LIN {X 0,Y 354.586,Z 442.804,A -85,B 0,C 180,E1 -14686.804,E2 -14686.804} C_VEL
LIN {X 0,Y 350.796,Z 438.924,A -85,B 0,C 180,E1 -14687.678,E2 -14687.678} C_VEL
LIN {X 0,Y 348.706,Z 436.523,A -85,B 0,C 180,E1 -14688.15,E2 -14688.15} C_VEL
LIN {X 0,Y 345.386,Z 432.719,A -85,B 0,C 180,E1 -14688.87,E2 -14688.87} C_VEL
LIN {X 0,Y 343.539,Z 430.553,A -85,B 0,C 180,E1 -14689.252,E2 -14689.252} C_VEL
LIN {X 0,Y 340.657,Z 426.868,A -85,B 0,C 180,E1 -14689.842,E2 -14689.842} C_VEL
LIN {X 0,Y 337.415,Z 422.834,A -85,B 0,C 180,E1 -14690.475,E2 -14690.475} C_VEL
LIN {X 0,Y 336.252,Z 421.04,A -85,B 0,C 180,E1 -14690.703,E2 -14690.703} C_VEL
LIN {X 0,Y 334.391,Z 418.724,A -85,B 0,C 180,E1 -14691.054,E2 -14691.054} C_VEL
LIN {X 0,Y 333.681,Z 416.421,A -85,B 0,C 180,E1 -14691.256,E2 -14691.256} C_VEL
LIN {X 0,Y 333.714,Z 416.415,A -85,B 0,C 180,E1 -14695.101,E2 -14695.101} C_VEL
LIN {X 0,Y 333.711,Z 416.417,A -85,B 0,C 180,E1 -14697.809,E2 -14697.809} C_VEL
LIN {X 0,Y 333.685,Z 416.417,A -85,B 0,C 180,E1 -14700.363,E2 -14700.363} C_VEL
LIN {X 0,Y 333.668,Z 416.419,A -85,B 0,C 180,E1 -14704.658,E2 -14704.658} C_VEL
LIN {X 0,Y 333.648,Z 416.425,A -85,B 0,C 180,E1 -14707.651,E2 -14707.651} C_VEL
LIN {X 0,Y 333.64,Z 416.423,A -85,B 0,C 180,E1 -14710.767,E2 -14710.767} C_VEL
LIN {X 0,Y 333.619,Z 416.425,A -85,B 0,C 180,E1 -14714.256,E2 -14714.256} C_VEL
LIN {X 0,Y 333.635,Z 416.425,A -85,B 0,C 180,E1 -14717.618,E2 -14717.618} C_VEL
LIN {X 0,Y 333.645,Z 416.427,A -85,B 0,C 180,E1 -14721.202,E2 -14721.202} C_VEL
LIN {X 0,Y 333.669,Z 416.419,A -85,B 0,C 180,E1 -14723.861,E2 -14723.861} C_VEL
LIN {X 0,Y 333.636,Z 416.425,A -85,B 0,C 180,E1 -14727.413,E2 -14727.413} C_VEL
LIN {X 0,Y 333.704,Z 416.42,A -85,B 0,C 180,E1 -14731.028,E2 -14731.028} C_VEL
LIN {X 0,Y 333.705,Z 416.417,A -85,B 0,C 180,E1 -14734.698,E2 -14734.698} C_VEL
LIN {X 0,Y 333.712,Z 416.413,A -85,B 0,C 180,E1 -14737.914,E2 -14737.914} C_VEL
LIN {X 0,Y 333.697,Z 416.414,A -85,B 0,C 180,E1 -14739.932,E2 -14739.932} C_VEL
LIN {X 0,Y 333.086,Z 416.496,A -85,B 0,C 180,E1 -14740.94,E2 -14740.94} C_VEL
LIN {X 0,Y 330.26,Z 416.849,A -85,B 0,C 180,E1 -14742.579,E2 -14742.579} C_VEL
LIN {X 0,Y 327.845,Z 417.15,A -85,B 0,C 180,E1 -14743.907,E2 -14743.907} C_VEL
LIN {X 0,Y 326.824,Z 417.275,A -85,B 0,C 180,E1 -14744.934,E2 -14744.934} C_VEL
LIN {X 0,Y 326.75,Z 417.281,A -85,B 0,C 180,E1 -14745.283,E2 -14745.283} C_VEL
LIN {X 0,Y 326.762,Z 417.283,A -85,B 0,C 180,E1 -14748.839,E2 -14748.839} C_VEL
LIN {X 0,Y 326.951,Z 417.26,A -85,B 0,C 180,E1 -14752.59,E2 -14752.59} C_VEL
LIN {X 0,Y 326.771,Z 417.278,A -85,B 0,C 180,E1 -14755.065,E2 -14755.065} C_VEL
LIN {X 0,Y 327.041,Z 417.239,A -85,B 0,C 180,E1 -14757.537,E2 -14757.537} C_VEL
LIN {X 0,Y 327.191,Z 417.223,A -85,B 0,C 180,E1 -14760.001,E2 -14760.001} C_VEL
LIN {X 0,Y 327.041,Z 417.249,A -85,B 0,C 180,E1 -14762.464,E2 -14762.464} C_VEL
LIN {X 0,Y 326.983,Z 417.255,A -85,B 0,C 180,E1 -14766.17,E2 -14766.17} C_VEL
LIN {X 0,Y 326.799,Z 417.276,A -85,B 0,C 180,E1 -14769.907,E2 -14769.907} C_VEL
LIN {X 0,Y 326.753,Z 417.281,A -85,B 0,C 180,E1 -14773.686,E2 -14773.686} C_VEL
LIN {X 0,Y 326.694,Z 417.288,A -85,B 0,C 180,E1 -14777.529,E2 -14777.529} C_VEL
LIN {X 0,Y 326.653,Z 417.298,A -85,B 0,C 180,E1 -14780.136,E2 -14780.136} C_VEL
LIN {X 0,Y 326.644,Z 417.3,A -85,B 0,C 180,E1 -14784.13,E2 -14784.13} C_VEL
LIN {X 0,Y 326.681,Z 417.29,A -85,B 0,C 180,E1 -14786.859,E2 -14786.859} C_VEL
LIN {X 0,Y 326.638,Z 417.298,A -85,B 0,C 180,E1 -14790.613,E2 -14790.613} C_VEL
LIN {X 0,Y 326.606,Z 417.305,A -85,B 0,C 180,E1 -14794.02,E2 -14794.02} C_VEL
LIN {X 0,Y 326.683,Z 417.655,A -85,B 0,C 180,E1 -14795.511,E2 -14795.511} C_VEL
LIN {X 0,Y 327.038,Z 420.312,A -85,B 0,C 180,E1 -14799.32,E2 -14799.32} C_VEL
LIN {X 0,Y 327.48,Z 423.224,A -85,B 0,C 180,E1 -14803.143,E2 -14803.143} C_VEL
LIN {X 0,Y 327.639,Z 424.827,A -85,B 0,C 180,E1 -14805.062,E2 -14805.062} C_VEL
LIN {X 0,Y 327.663,Z 427.715,A -85,B 0,C 180,E1 -14808.325,E2 -14808.325} C_VEL
LIN {X 0,Y 327.32,Z 430.741,A -85,B 0,C 180,E1 -14811.49,E2 -14811.49} C_VEL
LIN {X 0,Y 326.883,Z 434.094,A -85,B 0,C 180,E1 -14814.787,E2 -14814.787} C_VEL
LIN {X 0,Y 326.537,Z 436.909,A -85,B 0,C 180,E1 -14817.448,E2 -14817.448} C_VEL
LIN {X 0,Y 326.123,Z 440.042,A -85,B 0,C 180,E1 -14820.288,E2 -14820.288} C_VEL
LIN {X 0,Y 325.778,Z 443.169,A -85,B 0,C 180,E1 -14823.062,E2 -14823.062} C_VEL
LIN {X 0,Y 325.536,Z 446.331,A -85,B 0,C 180,E1 -14825.784,E2 -14825.784} C_VEL
LIN {X 0,Y 325.333,Z 448.523,A -85,B 0,C 180,E1 -14827.658,E2 -14827.658} C_VEL
LIN {X 0,Y 328.277,Z 460.951,A -85,B 0,C 180,E1 -14828.388,E2 -14828.388} C_VEL
LIN {X 0,Y 330.744,Z 474.544,A -85,B 0,C 180,E1 -14829.4,E2 -14829.4} C_VEL
LIN {X 0,Y 331.996,Z 485.066,A -85,B 0,C 180,E1 -14830.364,E2 -14830.364} C_VEL
LIN {X 0,Y 332.325,Z 489.987,A -85,B 0,C 180,E1 -14830.866,E2 -14830.866} C_VEL
LIN {X 0,Y 330.84,Z 502.177,A -85,B 0,C 180,E1 -14832.22,E2 -14832.22} C_VEL
LIN {X 0,Y 329.853,Z 509.927,A -85,B 0,C 180,E1 -14833.284,E2 -14833.284} C_VEL
LIN {X 0,Y 328.869,Z 517.509,A -85,B 0,C 180,E1 -14834.521,E2 -14834.521} C_VEL
LIN {X 0,Y 327.798,Z 525.266,A -85,B 0,C 180,E1 -14836.043,E2 -14836.043} C_VEL
LIN {X 0,Y 326.796,Z 531.801,A -85,B 0,C 180,E1 -14837.581,E2 -14837.581} C_VEL
LIN {X 0,Y 326.23,Z 536.304,A -85,B 0,C 180,E1 -14838.82,E2 -14838.82} C_VEL
LIN {X 0,Y 325.601,Z 541.798,A -85,B 0,C 180,E1 -14840.684,E2 -14840.684} C_VEL
LIN {X 0,Y 325.159,Z 546.124,A -85,B 0,C 180,E1 -14842.549,E2 -14842.549} C_VEL
LIN {X 0,Y 324.906,Z 549.205,A -85,B 0,C 180,E1 -14844.285,E2 -14844.285} C_VEL
LIN {X 0,Y 324.902,Z 551.682,A -85,B 0,C 180,E1 -14846.279,E2 -14846.279} C_VEL
LIN {X 0,Y 324.838,Z 552.74,A -85,B 0,C 180,E1 -14847.52,E2 -14847.52} C_VEL
LIN {X 0,Y 324.823,Z 553.329,A -85,B 0,C 180,E1 -14848.76,E2 -14848.76} C_VEL
LIN {X 0,Y 324.873,Z 553.485,A -85,B 0,C 180,E1 -14850,E2 -14850} C_VEL
LIN {X 0,Y 324.823,Z 553.329,A -85,B 0,C 180,E1 -14851.24,E2 -14851.24} C_VEL
LIN {X 0,Y 324.838,Z 552.74,A -85,B 0,C 180,E1 -14852.48,E2 -14852.48} C_VEL
LIN {X 0,Y 324.892,Z 550.292,A -85,B 0,C 180,E1 -14854.964,E2 -14854.964} C_VEL
LIN {X 0,Y 325.047,Z 547.341,A -85,B 0,C 180,E1 -14856.83,E2 -14856.83} C_VEL
LIN {X 0,Y 325.423,Z 543.352,A -85,B 0,C 180,E1 -14858.695,E2 -14858.695} C_VEL
LIN {X 0,Y 325.993,Z 538.221,A -85,B 0,C 180,E1 -14860.559,E2 -14860.559} C_VEL
LIN {X 0,Y 326.648,Z 532.957,A -85,B 0,C 180,E1 -14862.109,E2 -14862.109} C_VEL
LIN {X 0,Y 327.582,Z 526.642,A -85,B 0,C 180,E1 -14863.65,E2 -14863.65} C_VEL
LIN {X 0,Y 328.363,Z 520.689,A -85,B 0,C 180,E1 -14864.882,E2 -14864.882} C_VEL
LIN {X 0,Y 329.338,Z 513.197,A -85,B 0,C 180,E1 -14866.199,E2 -14866.199} C_VEL
LIN {X 0,Y 330.33,Z 505.58,A -85,B 0,C 180,E1 -14867.329,E2 -14867.329} C_VEL
LIN {X 0,Y 331.467,Z 497.071,A -85,B 0,C 180,E1 -14868.384,E2 -14868.384} C_VEL
LIN {X 0,Y 332.302,Z 489.987,A -85,B 0,C 180,E1 -14869.136,E2 -14869.136} C_VEL
LIN {X 0,Y 331.418,Z 479.637,A -85,B 0,C 180,E1 -14870.149,E2 -14870.149} C_VEL
LIN {X 0,Y 329.995,Z 469.715,A -85,B 0,C 180,E1 -14870.978,E2 -14870.978} C_VEL
LIN {X 0,Y 327.939,Z 459.393,A -85,B 0,C 180,E1 -14871.708,E2 -14871.708} C_VEL
LIN {X 0,Y 325.333,Z 448.523,A -85,B 0,C 180,E1 -14872.342,E2 -14872.342} C_VEL
LIN {X 0,Y 325.64,Z 444.744,A -85,B 0,C 180,E1 -14875.571,E2 -14875.571} C_VEL
LIN {X 0,Y 325.925,Z 441.591,A -85,B 0,C 180,E1 -14878.319,E2 -14878.319} C_VEL
LIN {X 0,Y 326.33,Z 438.464,A -85,B 0,C 180,E1 -14881.122,E2 -14881.122} C_VEL
LIN {X 0,Y 326.71,Z 435.355,A -85,B 0,C 180,E1 -14884.006,E2 -14884.006} C_VEL
LIN {X 0,Y 327.172,Z 431.885,A -85,B 0,C 180,E1 -14887.363,E2 -14887.363} C_VEL
LIN {X 0,Y 327.499,Z 429.209,A -85,B 0,C 180,E1 -14890.074,E2 -14890.074} C_VEL
LIN {X 0,Y 327.671,Z 426.322,A -85,B 0,C 180,E1 -14893.176,E2 -14893.176} C_VEL
LIN {X 0,Y 327.613,Z 424.686,A -85,B 0,C 180,E1 -14895.065,E2 -14895.065} C_VEL
LIN {X 0,Y 327.24,Z 421.707,A -85,B 0,C 180,E1 -14898.735,E2 -14898.735} C_VEL
LIN {X 0,Y 326.823,Z 418.85,A -85,B 0,C 180,E1 -14902.715,E2 -14902.715} C_VEL
LIN {X 0,Y 326.637,Z 417.429,A -85,B 0,C 180,E1 -14904.845,E2 -14904.845} C_VEL
LIN {X 0,Y 326.612,Z 417.303,A -85,B 0,C 180,E1 -14907.455,E2 -14907.455} C_VEL
LIN {X 0,Y 326.658,Z 417.295,A -85,B 0,C 180,E1 -14910.34,E2 -14910.34} C_VEL
LIN {X 0,Y 326.686,Z 417.29,A -85,B 0,C 180,E1 -14914.515,E2 -14914.515} C_VEL
LIN {X 0,Y 326.614,Z 417.299,A -85,B 0,C 180,E1 -14918.542,E2 -14918.542} C_VEL
LIN {X 0,Y 326.74,Z 417.283,A -85,B 0,C 180,E1 -14921.177,E2 -14921.177} C_VEL
LIN {X 0,Y 326.758,Z 417.283,A -85,B 0,C 180,E1 -14925.432,E2 -14925.432} C_VEL
LIN {X 0,Y 326.763,Z 417.279,A -85,B 0,C 180,E1 -14928.838,E2 -14928.838} C_VEL
LIN {X 0,Y 326.952,Z 417.255,A -85,B 0,C 180,E1 -14932.589,E2 -14932.589} C_VEL
LIN {X 0,Y 326.771,Z 417.28,A -85,B 0,C 180,E1 -14935.064,E2 -14935.064} C_VEL
LIN {X 0,Y 327.041,Z 417.249,A -85,B 0,C 180,E1 -14937.536,E2 -14937.536} C_VEL
LIN {X 0,Y 327.191,Z 417.223,A -85,B 0,C 180,E1 -14939.999,E2 -14939.999} C_VEL
LIN {X 0,Y 327.041,Z 417.239,A -85,B 0,C 180,E1 -14942.463,E2 -14942.463} C_VEL
LIN {X 0,Y 326.953,Z 417.255,A -85,B 0,C 180,E1 -14946.64,E2 -14946.64} C_VEL
LIN {X 0,Y 326.798,Z 417.275,A -85,B 0,C 180,E1 -14949.906,E2 -14949.906} C_VEL
LIN {X 0,Y 326.751,Z 417.281,A -85,B 0,C 180,E1 -14953.685,E2 -14953.685} C_VEL
LIN {X 0,Y 326.691,Z 417.29,A -85,B 0,C 180,E1 -14957.528,E2 -14957.528} C_VEL
LIN {X 0,Y 326.658,Z 417.291,A -85,B 0,C 180,E1 -14960.135,E2 -14960.135} C_VEL
LIN {X 0,Y 326.644,Z 417.293,A -85,B 0,C 180,E1 -14964.129,E2 -14964.129} C_VEL
LIN {X 0,Y 326.678,Z 417.293,A -85,B 0,C 180,E1 -14966.857,E2 -14966.857} C_VEL
LIN {X 0,Y 326.632,Z 417.298,A -85,B 0,C 180,E1 -14970.611,E2 -14970.611} C_VEL
LIN {X 0,Y 326.599,Z 417.299,A -85,B 0,C 180,E1 -14974.019,E2 -14974.019} C_VEL
LIN {X 0,Y 326.622,Z 417.299,A -85,B 0,C 180,E1 -14977.239,E2 -14977.239} C_VEL
LIN {X 0,Y 326.628,Z 417.297,A -85,B 0,C 180,E1 -14980.202,E2 -14980.202} C_VEL
LIN {X 0,Y 326.611,Z 417.298,A -85,B 0,C 180,E1 -14983.516,E2 -14983.516} C_VEL
LIN {X 0,Y 326.579,Z 417.305,A -85,B 0,C 180,E1 -14987.026,E2 -14987.026} C_VEL
LIN {X 0,Y 326.606,Z 417.303,A -85,B 0,C 180,E1 -14990.773,E2 -14990.773} C_VEL
LIN {X 0,Y 326.608,Z 417.304,A -85,B 0,C 180,E1 -14994.481,E2 -14994.481} C_VEL
LIN {X 0,Y 326.602,Z 417.3,A -85,B 0,C 180,E1 -14997.456,E2 -14997.456} C_VEL
LIN {X 0,Y 326.642,Z 417.299,A -85,B 0,C 180,E1 -15000.34,E2 -15000.34} C_VEL
LIN {X 0,Y 326.685,Z 417.294,A -85,B 0,C 180,E1 -15004.516,E2 -15004.516} C_VEL
LIN {X 0,Y 326.689,Z 417.462,A -85,B 0,C 180,E1 -15007.849,E2 -15007.849} C_VEL
LIN {X 0,Y 327.791,Z 420.343,A -85,B 0,C 180,E1 -15008.062,E2 -15008.062} C_VEL
LIN {X 0,Y 329.517,Z 422.626,A -85,B 0,C 180,E1 -15008.362,E2 -15008.362} C_VEL
LIN {X 0,Y 331.852,Z 425.984,A -85,B 0,C 180,E1 -15008.781,E2 -15008.781} C_VEL
LIN {X 0,Y 335.942,Z 431.221,A -85,B 0,C 180,E1 -15009.532,E2 -15009.532} C_VEL
LIN {X 0,Y 340.413,Z 436.599,A -85,B 0,C 180,E1 -15010.402,E2 -15010.402} C_VEL
LIN {X 0,Y 345.47,Z 442.395,A -85,B 0,C 180,E1 -15011.447,E2 -15011.447} C_VEL
LIN {X 0,Y 350.946,Z 448.281,A -85,B 0,C 180,E1 -15012.682,E2 -15012.682} C_VEL
LIN {X 0,Y 353.907,Z 451.302,A -85,B 0,C 180,E1 -15013.392,E2 -15013.392} C_VEL
LIN {X 0,Y 358.155,Z 455.445,A -85,B 0,C 180,E1 -15014.486,E2 -15014.486} C_VEL
LIN {X 0,Y 360.414,Z 457.588,A -85,B 0,C 180,E1 -15015.099,E2 -15015.099} C_VEL
LIN {X 0,Y 364.615,Z 461.693,A -85,B 0,C 180,E1 -15016.351,E2 -15016.351} C_VEL
LIN {X 0,Y 367.642,Z 464.194,A -85,B 0,C 180,E1 -15017.326,E2 -15017.326} C_VEL
LIN {X 0,Y 370.733,Z 467.391,A -85,B 0,C 180,E1 -15018.475,E2 -15018.475} C_VEL
LIN {X 0,Y 372.478,Z 468.776,A -85,B 0,C 180,E1 -15019.124,E2 -15019.124} C_VEL
LIN {X 0,Y 375.438,Z 470.677,A -85,B 0,C 180,E1 -15020.301,E2 -15020.301} C_VEL
LIN {X 0,Y 378.566,Z 473.961,A -85,B 0,C 180,E1 -15021.942,E2 -15021.942} C_VEL
LIN {X 0,Y 381.303,Z 476.371,A -85,B 0,C 180,E1 -15023.651,E2 -15023.651} C_VEL
LIN {X 0,Y 382.801,Z 477.354,A -85,B 0,C 180,E1 -15024.733,E2 -15024.733} C_VEL
LIN {X 0,Y 384.081,Z 477.889,A -85,B 0,C 180,E1 -15025.803,E2 -15025.803} C_VEL
LIN {X 0,Y 385.11,Z 478.153,A -85,B 0,C 180,E1 -15026.862,E2 -15026.862} C_VEL
LIN {X 0,Y 385.86,Z 478.305,A -85,B 0,C 180,E1 -15027.912,E2 -15027.912} C_VEL
LIN {X 0,Y 386.321,Z 478.391,A -85,B 0,C 180,E1 -15028.958,E2 -15028.958} C_VEL
LIN {X 0,Y 386.476,Z 478.443,A -85,B 0,C 180,E1 -15030,E2 -15030} C_VEL
LIN {X 0,Y 386.321,Z 478.386,A -85,B 0,C 180,E1 -15031.042,E2 -15031.042} C_VEL
LIN {X 0,Y 385.842,Z 478.34,A -85,B 0,C 180,E1 -15032.088,E2 -15032.088} C_VEL
LIN {X 0,Y 385.11,Z 478.141,A -85,B 0,C 180,E1 -15033.138,E2 -15033.138} C_VEL
LIN {X 0,Y 384.081,Z 477.915,A -85,B 0,C 180,E1 -15034.197,E2 -15034.197} C_VEL
LIN {X 0,Y 381.666,Z 476.606,A -85,B 0,C 180,E1 -15036.098,E2 -15036.098} C_VEL
LIN {X 0,Y 379.583,Z 474.969,A -85,B 0,C 180,E1 -15037.447,E2 -15037.447} C_VEL
LIN {X 0,Y 377.021,Z 472.248,A -85,B 0,C 180,E1 -15038.902,E2 -15038.902} C_VEL
LIN {X 0,Y 375.363,Z 470.65,A -85,B 0,C 180,E1 -15039.701,E2 -15039.701} C_VEL
LIN {X 0,Y 372.23,Z 468.586,A -85,B 0,C 180,E1 -15040.951,E2 -15040.951} C_VEL
LIN {X 0,Y 368.479,Z 465.181,A -85,B 0,C 180,E1 -15042.358,E2 -15042.358} C_VEL
LIN {X 0,Y 366.19,Z 462.867,A -85,B 0,C 180,E1 -15043.156,E2 -15043.156} C_VEL
LIN {X 0,Y 362.313,Z 459.671,A -85,B 0,C 180,E1 -15044.327,E2 -15044.327} C_VEL
LIN {X 0,Y 358.551,Z 455.713,A -85,B 0,C 180,E1 -15045.413,E2 -15045.413} C_VEL
LIN {X 0,Y 354.635,Z 452.162,A -85,B 0,C 180,E1 -15046.413,E2 -15046.413} C_VEL
LIN {X 0,Y 351.288,Z 448.602,A -85,B 0,C 180,E1 -15047.235,E2 -15047.235} C_VEL
LIN {X 0,Y 347.179,Z 444.187,A -85,B 0,C 180,E1 -15048.187,E2 -15048.187} C_VEL
LIN {X 0,Y 342.186,Z 438.709,A -85,B 0,C 180,E1 -15049.238,E2 -15049.238} C_VEL
LIN {X 0,Y 337.209,Z 432.791,A -85,B 0,C 180,E1 -15050.226,E2 -15050.226} C_VEL
LIN {X 0,Y 333.139,Z 427.618,A -85,B 0,C 180,E1 -15050.994,E2 -15050.994} C_VEL
LIN {X 0,Y 329.77,Z 423.148,A -85,B 0,C 180,E1 -15051.586,E2 -15051.586} C_VEL
LIN {X 0,Y 328.729,Z 421.468,A -85,B 0,C 180,E1 -15051.779,E2 -15051.779} C_VEL
LIN {X 0,Y 327.095,Z 418.984,A -85,B 0,C 180,E1 -15052.062,E2 -15052.062} C_VEL
LIN {X 0,Y 326.675,Z 417.293,A -85,B 0,C 180,E1 -15052.178,E2 -15052.178} C_VEL
LIN {X 0,Y 326.685,Z 417.294,A -85,B 0,C 180,E1 -15055.484,E2 -15055.484} C_VEL
LIN {X 0,Y 326.642,Z 417.299,A -85,B 0,C 180,E1 -15059.66,E2 -15059.66} C_VEL
LIN {X 0,Y 326.601,Z 417.301,A -85,B 0,C 180,E1 -15064.019,E2 -15064.019} C_VEL
LIN {X 0,Y 326.623,Z 417.301,A -85,B 0,C 180,E1 -15067.239,E2 -15067.239} C_VEL
LIN {X 0,Y 326.572,Z 417.307,A -85,B 0,C 180,E1 -15071.131,E2 -15071.131} C_VEL
LIN {X 0,Y 326.55,Z 417.307,A -85,B 0,C 180,E1 -15074.748,E2 -15074.748} C_VEL
LIN {X 0,Y 326.569,Z 417.303,A -85,B 0,C 180,E1 -15078.154,E2 -15078.154} C_VEL
LIN {X 0,Y 326.591,Z 417.304,A -85,B 0,C 180,E1 -15081.388,E2 -15081.388} C_VEL
LIN {X 0,Y 326.612,Z 417.301,A -85,B 0,C 180,E1 -15084.851,E2 -15084.851} C_VEL
LIN {X 0,Y 326.6,Z 417.302,A -85,B 0,C 180,E1 -15087.456,E2 -15087.456} C_VEL
LIN {X 0,Y 326.653,Z 417.293,A -85,B 0,C 180,E1 -15090.341,E2 -15090.341} C_VEL
LIN {X 0,Y 326.683,Z 417.291,A -85,B 0,C 180,E1 -15094.516,E2 -15094.516} C_VEL
LIN {X 0,Y 326.641,Z 417.297,A -85,B 0,C 180,E1 -15098.546,E2 -15098.546} C_VEL
LIN {X 0,Y 326.737,Z 417.285,A -85,B 0,C 180,E1 -15101.178,E2 -15101.178} C_VEL
LIN {X 0,Y 326.75,Z 417.281,A -85,B 0,C 180,E1 -15105.283,E2 -15105.283} C_VEL
LIN {X 0,Y 326.1,Z 417.364,A -85,B 0,C 180,E1 -15106.312,E2 -15106.312} C_VEL
LIN {X 0,Y 323.233,Z 417.719,A -85,B 0,C 180,E1 -15107.986,E2 -15107.986} C_VEL
LIN {X 0,Y 320.824,Z 418.019,A -85,B 0,C 180,E1 -15109.343,E2 -15109.343} C_VEL
LIN {X 0,Y 319.839,Z 418.143,A -85,B 0,C 180,E1 -15110.393,E2 -15110.393} C_VEL
LIN {X 0,Y 319.786,Z 418.147,A -85,B 0,C 180,E1 -15110.749,E2 -15110.749} C_VEL
LIN {X 0,Y 319.937,Z 418.129,A -85,B 0,C 180,E1 -15113.695,E2 -15113.695} C_VEL
LIN {X 0,Y 319.985,Z 418.117,A -85,B 0,C 180,E1 -15117.483,E2 -15117.483} C_VEL
LIN {X 0,Y 320.143,Z 418.101,A -85,B 0,C 180,E1 -15120.001,E2 -15120.001} C_VEL
LIN {X 0,Y 319.985,Z 418.129,A -85,B 0,C 180,E1 -15122.518,E2 -15122.518} C_VEL
LIN {X 0,Y 319.937,Z 418.134,A -85,B 0,C 180,E1 -15126.306,E2 -15126.306} C_VEL
LIN {X 0,Y 319.831,Z 418.145,A -85,B 0,C 180,E1 -15128.849,E2 -15128.849} C_VEL
LIN {X 0,Y 319.676,Z 418.165,A -85,B 0,C 180,E1 -15132.701,E2 -15132.701} C_VEL
LIN {X 0,Y 319.694,Z 418.16,A -85,B 0,C 180,E1 -15135.296,E2 -15135.296} C_VEL
LIN {X 0,Y 319.647,Z 418.166,A -85,B 0,C 180,E1 -15139.257,E2 -15139.257} C_VEL
LIN {X 0,Y 319.556,Z 418.178,A -85,B 0,C 180,E1 -15143.321,E2 -15143.321} C_VEL
LIN {X 0,Y 319.631,Z 418.174,A -85,B 0,C 180,E1 -15146.089,E2 -15146.089} C_VEL
LIN {X 0,Y 319.586,Z 418.174,A -85,B 0,C 180,E1 -15148.935,E2 -15148.935} C_VEL
LIN {X 0,Y 319.535,Z 418.186,A -85,B 0,C 180,E1 -15151.862,E2 -15151.862} C_VEL
LIN {X 0,Y 319.587,Z 418.38,A -85,B 0,C 180,E1 -15154.874,E2 -15154.874} C_VEL
LIN {X 0,Y 319.876,Z 420.418,A -85,B 0,C 180,E1 -15157.966,E2 -15157.966} C_VEL
LIN {X 0,Y 320.298,Z 423.169,A -85,B 0,C 180,E1 -15161.754,E2 -15161.754} C_VEL
LIN {X 0,Y 320.561,Z 425.375,A -85,B 0,C 180,E1 -15164.554,E2 -15164.554} C_VEL
LIN {X 0,Y 320.623,Z 428.509,A -85,B 0,C 180,E1 -15168.183,E2 -15168.183} C_VEL
LIN {X 0,Y 320.39,Z 430.649,A -85,B 0,C 180,E1 -15170.497,E2 -15170.497} C_VEL
LIN {X 0,Y 319.862,Z 434.465,A -85,B 0,C 180,E1 -15174.387,E2 -15174.387} C_VEL
LIN {X 0,Y 319.354,Z 438.337,A -85,B 0,C 180,E1 -15178.119,E2 -15178.119} C_VEL
LIN {X 0,Y 318.837,Z 442.385,A -85,B 0,C 180,E1 -15181.85,E2 -15181.85} C_VEL
LIN {X 0,Y 318.509,Z 446.169,A -85,B 0,C 180,E1 -15185.214,E2 -15185.214} C_VEL
LIN {X 0,Y 318.289,Z 448.358,A -85,B 0,C 180,E1 -15187.142,E2 -15187.142} C_VEL
LIN {X 0,Y 320.761,Z 458.319,A -85,B 0,C 180,E1 -15187.739,E2 -15187.739} C_VEL
LIN {X 0,Y 322.765,Z 468.257,A -85,B 0,C 180,E1 -15188.448,E2 -15188.448} C_VEL
LIN {X 0,Y 324.316,Z 478.331,A -85,B 0,C 180,E1 -15189.3,E2 -15189.3} C_VEL
LIN {X 0,Y 325.376,Z 488.146,A -85,B 0,C 180,E1 -15190.276,E2 -15190.276} C_VEL
LIN {X 0,Y 325.336,Z 492.821,A -85,B 0,C 180,E1 -15190.766,E2 -15190.766} C_VEL
LIN {X 0,Y 323.912,Z 503.114,A -85,B 0,C 180,E1 -15191.99,E2 -15191.99} C_VEL
LIN {X 0,Y 322.75,Z 511.645,A -85,B 0,C 180,E1 -15193.231,E2 -15193.231} C_VEL
LIN {X 0,Y 321.72,Z 519.073,A -85,B 0,C 180,E1 -15194.52,E2 -15194.52} C_VEL
LIN {X 0,Y 320.895,Z 525.068,A -85,B 0,C 180,E1 -15195.736,E2 -15195.736} C_VEL
LIN {X 0,Y 319.847,Z 531.604,A -85,B 0,C 180,E1 -15197.307,E2 -15197.307} C_VEL
LIN {X 0,Y 319.221,Z 536.106,A -85,B 0,C 180,E1 -15198.572,E2 -15198.572} C_VEL
LIN {X 0,Y 318.582,Z 541.601,A -85,B 0,C 180,E1 -15200.477,E2 -15200.477} C_VEL
LIN {X 0,Y 318.087,Z 545.926,A -85,B 0,C 180,E1 -15202.382,E2 -15202.382} C_VEL
LIN {X 0,Y 317.807,Z 549.28,A -85,B 0,C 180,E1 -15204.35,E2 -15204.35} C_VEL
LIN {X 0,Y 317.809,Z 551.485,A -85,B 0,C 180,E1 -15206.196,E2 -15206.196} C_VEL
LIN {X 0,Y 317.76,Z 552.543,A -85,B 0,C 180,E1 -15207.465,E2 -15207.465} C_VEL
LIN {X 0,Y 317.735,Z 553.132,A -85,B 0,C 180,E1 -15208.733,E2 -15208.733} C_VEL
LIN {X 0,Y 317.735,Z 553.132,A -85,B 0,C 180,E1 -15211.267,E2 -15211.267} C_VEL
LIN {X 0,Y 317.76,Z 552.543,A -85,B 0,C 180,E1 -15212.535,E2 -15212.535} C_VEL
LIN {X 0,Y 317.806,Z 550.095,A -85,B 0,C 180,E1 -15215.075,E2 -15215.075} C_VEL
LIN {X 0,Y 317.986,Z 547.143,A -85,B 0,C 180,E1 -15216.982,E2 -15216.982} C_VEL
LIN {X 0,Y 318.382,Z 543.154,A -85,B 0,C 180,E1 -15218.889,E2 -15218.889} C_VEL
LIN {X 0,Y 318.978,Z 538.023,A -85,B 0,C 180,E1 -15220.794,E2 -15220.794} C_VEL
LIN {X 0,Y 319.659,Z 532.759,A -85,B 0,C 180,E1 -15222.378,E2 -15222.378} C_VEL
LIN {X 0,Y 320.677,Z 526.444,A -85,B 0,C 180,E1 -15223.95,E2 -15223.95} C_VEL
LIN {X 0,Y 321.48,Z 520.491,A -85,B 0,C 180,E1 -15225.208,E2 -15225.208} C_VEL
LIN {X 0,Y 322.41,Z 513.562,A -85,B 0,C 180,E1 -15226.462,E2 -15226.462} C_VEL
LIN {X 0,Y 323.543,Z 505.382,A -85,B 0,C 180,E1 -15227.704,E2 -15227.704} C_VEL
LIN {X 0,Y 324.73,Z 496.873,A -85,B 0,C 180,E1 -15228.779,E2 -15228.779} C_VEL
LIN {X 0,Y 325.467,Z 489.786,A -85,B 0,C 180,E1 -15229.554,E2 -15229.554} C_VEL
LIN {X 0,Y 324.446,Z 479.431,A -85,B 0,C 180,E1 -15230.602,E2 -15230.602} C_VEL
LIN {X 0,Y 323.039,Z 469.861,A -85,B 0,C 180,E1 -15231.429,E2 -15231.429} C_VEL
LIN {X 0,Y 320.94,Z 459.08,A -85,B 0,C 180,E1 -15232.212,E2 -15232.212} C_VEL
LIN {X 0,Y 318.291,Z 448.354,A -85,B 0,C 180,E1 -15232.861,E2 -15232.861} C_VEL
LIN {X 0,Y 318.597,Z 444.572,A -85,B 0,C 180,E1 -15236.179,E2 -15236.179} C_VEL
LIN {X 0,Y 319.189,Z 439.889,A -85,B 0,C 180,E1 -15240.425,E2 -15240.425} C_VEL
LIN {X 0,Y 319.558,Z 436.778,A -85,B 0,C 180,E1 -15243.354,E2 -15243.354} C_VEL
LIN {X 0,Y 319.968,Z 433.698,A -85,B 0,C 180,E1 -15246.373,E2 -15246.373} C_VEL
LIN {X 0,Y 320.448,Z 430.307,A -85,B 0,C 180,E1 -15249.859,E2 -15249.859} C_VEL
LIN {X 0,Y 320.617,Z 427.619,A -85,B 0,C 180,E1 -15252.805,E2 -15252.805} C_VEL
LIN {X 0,Y 320.542,Z 425.38,A -85,B 0,C 180,E1 -15255.443,E2 -15255.443} C_VEL
LIN {X 0,Y 320.235,Z 422.719,A -85,B 0,C 180,E1 -15258.822,E2 -15258.822} C_VEL
LIN {X 0,Y 319.85,Z 420.25,A -85,B 0,C 180,E1 -15262.279,E2 -15262.279} C_VEL
LIN {X 0,Y 319.586,Z 418.38,A -85,B 0,C 180,E1 -15265.126,E2 -15265.126} C_VEL
LIN {X 0,Y 319.535,Z 418.186,A -85,B 0,C 180,E1 -15268.138,E2 -15268.138} C_VEL
LIN {X 0,Y 319.613,Z 418.174,A -85,B 0,C 180,E1 -15271.587,E2 -15271.587} C_VEL
LIN {X 0,Y 319.598,Z 418.173,A -85,B 0,C 180,E1 -15275.303,E2 -15275.303} C_VEL
LIN {X 0,Y 319.597,Z 418.175,A -85,B 0,C 180,E1 -15279.399,E2 -15279.399} C_VEL
LIN {X 0,Y 319.653,Z 418.168,A -85,B 0,C 180,E1 -15282.072,E2 -15282.072} C_VEL
LIN {X 0,Y 319.726,Z 418.159,A -85,B 0,C 180,E1 -15286.007,E2 -15286.007} C_VEL
LIN {X 0,Y 319.746,Z 418.157,A -85,B 0,C 180,E1 -15289.872,E2 -15289.872} C_VEL
LIN {X 0,Y 319.906,Z 418.133,A -85,B 0,C 180,E1 -15292.425,E2 -15292.425} C_VEL
LIN {X 0,Y 319.74,Z 418.155,A -85,B 0,C 180,E1 -15294.955,E2 -15294.955} C_VEL
LIN {X 0,Y 319.985,Z 418.129,A -85,B 0,C 180,E1 -15297.482,E2 -15297.482} C_VEL
LIN {X 0,Y 320.143,Z 418.101,A -85,B 0,C 180,E1 -15299.999,E2 -15299.999} C_VEL
LIN {X 0,Y 319.985,Z 418.117,A -85,B 0,C 180,E1 -15302.517,E2 -15302.517} C_VEL
LIN {X 0,Y 319.914,Z 418.131,A -85,B 0,C 180,E1 -15306.628,E2 -15306.628} C_VEL
LIN {X 0,Y 319.745,Z 418.152,A -85,B 0,C 180,E1 -15310.127,E2 -15310.127} C_VEL
LIN {X 0,Y 319.723,Z 418.156,A -85,B 0,C 180,E1 -15314.724,E2 -15314.724} C_VEL
LIN {X 0,Y 319.682,Z 418.166,A -85,B 0,C 180,E1 -15319.037,E2 -15319.037} C_VEL
LIN {X 0,Y 319.562,Z 418.179,A -85,B 0,C 180,E1 -15323.319,E2 -15323.319} C_VEL
LIN {X 0,Y 319.628,Z 418.167,A -85,B 0,C 180,E1 -15326.088,E2 -15326.088} C_VEL
LIN {X 0,Y 319.583,Z 418.178,A -85,B 0,C 180,E1 -15328.933,E2 -15328.933} C_VEL
LIN {X 0,Y 319.525,Z 418.181,A -85,B 0,C 180,E1 -15331.862,E2 -15331.862} C_VEL
LIN {X 0,Y 319.573,Z 418.175,A -85,B 0,C 180,E1 -15335.543,E2 -15335.543} C_VEL
LIN {X 0,Y 319.577,Z 418.174,A -85,B 0,C 180,E1 -15338.006,E2 -15338.006} C_VEL
LIN {X 0,Y 319.589,Z 418.173,A -85,B 0,C 180,E1 -15341.611,E2 -15341.611} C_VEL
LIN {X 0,Y 319.557,Z 418.178,A -85,B 0,C 180,E1 -15345.271,E2 -15345.271} C_VEL
LIN {X 0,Y 319.523,Z 418.186,A -85,B 0,C 180,E1 -15348.712,E2 -15348.712} C_VEL
LIN {X 0,Y 319.572,Z 418.178,A -85,B 0,C 180,E1 -15352.344,E2 -15352.344} C_VEL
LIN {X 0,Y 319.554,Z 418.179,A -85,B 0,C 180,E1 -15355.124,E2 -15355.124} C_VEL
LIN {X 0,Y 319.561,Z 418.178,A -85,B 0,C 180,E1 -15359.059,E2 -15359.059} C_VEL
LIN {X 0,Y 319.601,Z 418.177,A -85,B 0,C 180,E1 -15362.498,E2 -15362.498} C_VEL
LIN {X 0,Y 319.6,Z 418.173,A -85,B 0,C 180,E1 -15365.304,E2 -15365.304} C_VEL
LIN {X 0,Y 319.568,Z 418.178,A -85,B 0,C 180,E1 -15367.016,E2 -15367.016} C_VEL
LIN {X 0,Y 320.699,Z 421.219,A -85,B 0,C 180,E1 -15367.234,E2 -15367.234} C_VEL
LIN {X 0,Y 322.178,Z 423.39,A -85,B 0,C 180,E1 -15367.456,E2 -15367.456} C_VEL
LIN {X 0,Y 324.618,Z 426.854,A -85,B 0,C 180,E1 -15367.845,E2 -15367.845} C_VEL
LIN {X 0,Y 327.332,Z 430.833,A -85,B 0,C 180,E1 -15368.295,E2 -15368.295} C_VEL
LIN {X 0,Y 332.3,Z 436.967,A -85,B 0,C 180,E1 -15369.178,E2 -15369.178} C_VEL
LIN {X 0,Y 336.681,Z 442.211,A -85,B 0,C 180,E1 -15370.02,E2 -15370.02} C_VEL
LIN {X 0,Y 342.128,Z 448.384,A -85,B 0,C 180,E1 -15371.144,E2 -15371.144} C_VEL
LIN {X 0,Y 347.568,Z 454.275,A -85,B 0,C 180,E1 -15372.384,E2 -15372.384} C_VEL
LIN {X 0,Y 350.27,Z 456.985,A -85,B 0,C 180,E1 -15373.028,E2 -15373.028} C_VEL
LIN {X 0,Y 354.736,Z 461.402,A -85,B 0,C 180,E1 -15374.183,E2 -15374.183} C_VEL
LIN {X 0,Y 356.911,Z 463.4,A -85,B 0,C 180,E1 -15374.764,E2 -15374.764} C_VEL
LIN {X 0,Y 361.783,Z 468.175,A -85,B 0,C 180,E1 -15376.237,E2 -15376.237} C_VEL
LIN {X 0,Y 364.702,Z 470.652,A -85,B 0,C 180,E1 -15377.166,E2 -15377.166} C_VEL
LIN {X 0,Y 367.994,Z 473.916,A -85,B 0,C 180,E1 -15378.388,E2 -15378.388} C_VEL
LIN {X 0,Y 371.43,Z 476.373,A -85,B 0,C 180,E1 -15379.706,E2 -15379.706} C_VEL
LIN {X 0,Y 373.7,Z 478.215,A -85,B 0,C 180,E1 -15380.715,E2 -15380.715} C_VEL
LIN {X 0,Y 376.798,Z 481.516,A -85,B 0,C 180,E1 -15382.498,E2 -15382.498} C_VEL
LIN {X 0,Y 378.545,Z 482.878,A -85,B 0,C 180,E1 -15383.604,E2 -15383.604} C_VEL
LIN {X 0,Y 380.799,Z 484.19,A -85,B 0,C 180,E1 -15385.278,E2 -15385.278} C_VEL
LIN {X 0,Y 382.437,Z 484.73,A -85,B 0,C 180,E1 -15386.84,E2 -15386.84} C_VEL
LIN {X 0,Y 383.22,Z 484.886,A -85,B 0,C 180,E1 -15387.898,E2 -15387.898} C_VEL
LIN {X 0,Y 383.694,Z 484.977,A -85,B 0,C 180,E1 -15388.95,E2 -15388.95} C_VEL
LIN {X 0,Y 383.856,Z 485.015,A -85,B 0,C 180,E1 -15390,E2 -15390} C_VEL
LIN {X 0,Y 383.694,Z 484.975,A -85,B 0,C 180,E1 -15391.05,E2 -15391.05} C_VEL
LIN {X 0,Y 383.199,Z 484.924,A -85,B 0,C 180,E1 -15392.102,E2 -15392.102} C_VEL
LIN {X 0,Y 382.437,Z 484.725,A -85,B 0,C 180,E1 -15393.16,E2 -15393.16} C_VEL
LIN {X 0,Y 380.795,Z 484.217,A -85,B 0,C 180,E1 -15394.714,E2 -15394.714} C_VEL
LIN {X 0,Y 378.523,Z 482.905,A -85,B 0,C 180,E1 -15396.396,E2 -15396.396} C_VEL
LIN {X 0,Y 376.092,Z 480.748,A -85,B 0,C 180,E1 -15397.949,E2 -15397.949} C_VEL
LIN {X 0,Y 372.658,Z 477.218,A -85,B 0,C 180,E1 -15399.772,E2 -15399.772} C_VEL
LIN {X 0,Y 369.698,Z 475.3,A -85,B 0,C 180,E1 -15400.958,E2 -15400.958} C_VEL
LIN {X 0,Y 366.474,Z 472.535,A -85,B 0,C 180,E1 -15402.178,E2 -15402.178} C_VEL
LIN {X 0,Y 361.772,Z 468.171,A -85,B 0,C 180,E1 -15403.756,E2 -15403.756} C_VEL
LIN {X 0,Y 358.426,Z 465.094,A -85,B 0,C 180,E1 -15404.768,E2 -15404.768} C_VEL
LIN {X 0,Y 355.426,Z 461.932,A -85,B 0,C 180,E1 -15405.64,E2 -15405.64} C_VEL
LIN {X 0,Y 351.147,Z 457.996,A -85,B 0,C 180,E1 -15406.74,E2 -15406.74} C_VEL
LIN {X 0,Y 347.688,Z 454.344,A -85,B 0,C 180,E1 -15407.593,E2 -15407.593} C_VEL
LIN {X 0,Y 343.361,Z 449.661,A -85,B 0,C 180,E1 -15408.589,E2 -15408.589} C_VEL
LIN {X 0,Y 338.348,Z 444.214,A -85,B 0,C 180,E1 -15409.639,E2 -15409.639} C_VEL
LIN {X 0,Y 333.053,Z 437.887,A -85,B 0,C 180,E1 -15410.682,E2 -15410.682} C_VEL
LIN {X 0,Y 329.035,Z 432.94,A -85,B 0,C 180,E1 -15411.412,E2 -15411.412} C_VEL
LIN {X 0,Y 325.098,Z 427.713,A -85,B 0,C 180,E1 -15412.079,E2 -15412.079} C_VEL
LIN {X 0,Y 322.182,Z 423.314,A -85,B 0,C 180,E1 -15412.546,E2 -15412.546} C_VEL
LIN {X 0,Y 319.965,Z 419.764,A -85,B 0,C 180,E1 -15412.879,E2 -15412.879} C_VEL
LIN {X 0,Y 319.584,Z 418.194,A -85,B 0,C 180,E1 -15412.96,E2 -15412.96} C_VEL
LIN {X 0,Y 319.629,Z 418.17,A -85,B 0,C 180,E1 -15416.088,E2 -15416.088} C_VEL
LIN {X 0,Y 319.574,Z 418.176,A -85,B 0,C 180,E1 -15418.934,E2 -15418.934} C_VEL
LIN {X 0,Y 319.525,Z 418.184,A -85,B 0,C 180,E1 -15421.862,E2 -15421.862} C_VEL
LIN {X 0,Y 319.575,Z 418.179,A -85,B 0,C 180,E1 -15425.543,E2 -15425.543} C_VEL
LIN {X 0,Y 319.568,Z 418.177,A -85,B 0,C 180,E1 -15428.008,E2 -15428.008} C_VEL
LIN {X 0,Y 319.52,Z 418.185,A -85,B 0,C 180,E1 -15431.597,E2 -15431.597} C_VEL
LIN {X 0,Y 319.509,Z 418.184,A -85,B 0,C 180,E1 -15434.738,E2 -15434.738} C_VEL
LIN {X 0,Y 319.554,Z 418.181,A -85,B 0,C 180,E1 -15437.018,E2 -15437.018} C_VEL
LIN {X 0,Y 319.54,Z 418.179,A -85,B 0,C 180,E1 -15440.371,E2 -15440.371} C_VEL
LIN {X 0,Y 319.572,Z 418.175,A -85,B 0,C 180,E1 -15444.457,E2 -15444.457} C_VEL
LIN {X 0,Y 319.525,Z 418.181,A -85,B 0,C 180,E1 -15448.138,E2 -15448.138} C_VEL
LIN {X 0,Y 319.609,Z 418.171,A -85,B 0,C 180,E1 -15451.589,E2 -15451.589} C_VEL
LIN {X 0,Y 319.597,Z 418.173,A -85,B 0,C 180,E1 -15455.304,E2 -15455.304} C_VEL
LIN {X 0,Y 319.59,Z 418.173,A -85,B 0,C 180,E1 -15458.048,E2 -15458.048} C_VEL
LIN {X 0,Y 319.682,Z 418.166,A -85,B 0,C 180,E1 -15460.963,E2 -15460.963} C_VEL
LIN {X 0,Y 319.723,Z 418.156,A -85,B 0,C 180,E1 -15465.276,E2 -15465.276} C_VEL
LIN {X 0,Y 319.745,Z 418.152,A -85,B 0,C 180,E1 -15469.873,E2 -15469.873} C_VEL
LIN {X 0,Y 319.786,Z 418.147,A -85,B 0,C 180,E1 -15470.749,E2 -15470.749} C_VEL
LIN {X 0,Y 319.51,Z 418.184,A -85,B 0,C 180,E1 -15471.452,E2 -15471.452} C_VEL
LIN {X 0,Y 317.54,Z 418.436,A -85,B 0,C 180,E1 -15472.831,E2 -15472.831} C_VEL
LIN {X 0,Y 313.742,Z 418.908,A -85,B 0,C 180,E1 -15474.896,E2 -15474.896} C_VEL
LIN {X 0,Y 312.753,Z 419.025,A -85,B 0,C 180,E1 -15475.971,E2 -15475.971} C_VEL
LIN {X 0,Y 312.716,Z 419.026,A -85,B 0,C 180,E1 -15476.335,E2 -15476.335} C_VEL
LIN {X 0,Y 312.984,Z 418.992,A -85,B 0,C 180,E1 -15478.714,E2 -15478.714} C_VEL
LIN {X 0,Y 312.984,Z 418.995,A -85,B 0,C 180,E1 -15481.287,E2 -15481.287} C_VEL
LIN {X 0,Y 312.71,Z 419.03,A -85,B 0,C 180,E1 -15485.158,E2 -15485.158} C_VEL
LIN {X 0,Y 312.847,Z 419.013,A -85,B 0,C 180,E1 -15487.747,E2 -15487.747} C_VEL
LIN {X 0,Y 312.663,Z 419.037,A -85,B 0,C 180,E1 -15491.672,E2 -15491.672} C_VEL
LIN {X 0,Y 312.695,Z 419.033,A -85,B 0,C 180,E1 -15494.888,E2 -15494.888} C_VEL
LIN {X 0,Y 312.604,Z 419.043,A -85,B 0,C 180,E1 -15499.226,E2 -15499.226} C_VEL
LIN {X 0,Y 312.521,Z 419.055,A -85,B 0,C 180,E1 -15502.781,E2 -15502.781} C_VEL
LIN {X 0,Y 312.599,Z 419.049,A -85,B 0,C 180,E1 -15505.937,E2 -15505.937} C_VEL
LIN {X 0,Y 312.543,Z 419.054,A -85,B 0,C 180,E1 -15509.651,E2 -15509.651} C_VEL
LIN {X 0,Y 312.522,Z 419.06,A -85,B 0,C 180,E1 -15513.691,E2 -15513.691} C_VEL
LIN {X 0,Y 312.518,Z 419.096,A -85,B 0,C 180,E1 -15514.209,E2 -15514.209} C_VEL
LIN {X 0,Y 312.868,Z 421.651,A -85,B 0,C 180,E1 -15518.169,E2 -15518.169} C_VEL
LIN {X 0,Y 313.134,Z 423.361,A -85,B 0,C 180,E1 -15520.609,E2 -15520.609} C_VEL
LIN {X 0,Y 313.496,Z 426.072,A -85,B 0,C 180,E1 -15524.163,E2 -15524.163} C_VEL
LIN {X 0,Y 313.572,Z 429.067,A -85,B 0,C 180,E1 -15527.75,E2 -15527.75} C_VEL
LIN {X 0,Y 313.45,Z 430.763,A -85,B 0,C 180,E1 -15529.671,E2 -15529.671} C_VEL
LIN {X 0,Y 313.039,Z 433.598,A -85,B 0,C 180,E1 -15532.688,E2 -15532.688} C_VEL
LIN {X 0,Y 312.535,Z 437.169,A -85,B 0,C 180,E1 -15536.308,E2 -15536.308} C_VEL
LIN {X 0,Y 312.208,Z 439.766,A -85,B 0,C 180,E1 -15538.82,E2 -15538.82} C_VEL
LIN {X 0,Y 311.583,Z 444.43,A -85,B 0,C 180,E1 -15543.185,E2 -15543.185} C_VEL
LIN {X 0,Y 311.28,Z 448.354,A -85,B 0,C 180,E1 -15546.608,E2 -15546.608} C_VEL
LIN {X 0,Y 313.613,Z 457.678,A -85,B 0,C 180,E1 -15547.182,E2 -15547.182} C_VEL
LIN {X 0,Y 315.528,Z 466.444,A -85,B 0,C 180,E1 -15547.822,E2 -15547.822} C_VEL
LIN {X 0,Y 317.048,Z 475.653,A -85,B 0,C 180,E1 -15548.595,E2 -15548.595} C_VEL
LIN {X 0,Y 318.155,Z 484.657,A -85,B 0,C 180,E1 -15549.472,E2 -15549.472} C_VEL
LIN {X 0,Y 318.604,Z 492.623,A -85,B 0,C 180,E1 -15550.343,E2 -15550.343} C_VEL
LIN {X 0,Y 317.148,Z 502.917,A -85,B 0,C 180,E1 -15551.593,E2 -15551.593} C_VEL
LIN {X 0,Y 315.919,Z 511.447,A -85,B 0,C 180,E1 -15552.857,E2 -15552.857} C_VEL
LIN {X 0,Y 314.846,Z 519.038,A -85,B 0,C 180,E1 -15554.207,E2 -15554.207} C_VEL
LIN {X 0,Y 313.76,Z 526.246,A -85,B 0,C 180,E1 -15555.736,E2 -15555.736} C_VEL
LIN {X 0,Y 312.696,Z 532.561,A -85,B 0,C 180,E1 -15557.342,E2 -15557.342} C_VEL
LIN {X 0,Y 311.975,Z 537.825,A -85,B 0,C 180,E1 -15558.961,E2 -15558.961} C_VEL
LIN {X 0,Y 311.359,Z 542.957,A -85,B 0,C 180,E1 -15560.909,E2 -15560.909} C_VEL
LIN {X 0,Y 310.921,Z 546.946,A -85,B 0,C 180,E1 -15562.859,E2 -15562.859} C_VEL
LIN {X 0,Y 310.703,Z 549.897,A -85,B 0,C 180,E1 -15564.809,E2 -15564.809} C_VEL
LIN {X 0,Y 310.683,Z 552.347,A -85,B 0,C 180,E1 -15567.407,E2 -15567.407} C_VEL
LIN {X 0,Y 310.65,Z 552.936,A -85,B 0,C 180,E1 -15568.704,E2 -15568.704} C_VEL
LIN {X 0,Y 310.65,Z 552.936,A -85,B 0,C 180,E1 -15571.296,E2 -15571.296} C_VEL
LIN {X 0,Y 310.683,Z 552.347,A -85,B 0,C 180,E1 -15572.593,E2 -15572.593} C_VEL
LIN {X 0,Y 310.709,Z 549.897,A -85,B 0,C 180,E1 -15575.191,E2 -15575.191} C_VEL
LIN {X 0,Y 310.921,Z 546.946,A -85,B 0,C 180,E1 -15577.141,E2 -15577.141} C_VEL
LIN {X 0,Y 311.359,Z 542.957,A -85,B 0,C 180,E1 -15579.091,E2 -15579.091} C_VEL
LIN {X 0,Y 311.975,Z 537.825,A -85,B 0,C 180,E1 -15581.039,E2 -15581.039} C_VEL
LIN {X 0,Y 312.696,Z 532.561,A -85,B 0,C 180,E1 -15582.658,E2 -15582.658} C_VEL
LIN {X 0,Y 313.764,Z 526.247,A -85,B 0,C 180,E1 -15584.264,E2 -15584.264} C_VEL
LIN {X 0,Y 314.824,Z 519.079,A -85,B 0,C 180,E1 -15585.786,E2 -15585.786} C_VEL
LIN {X 0,Y 315.879,Z 511.445,A -85,B 0,C 180,E1 -15587.145,E2 -15587.145} C_VEL
LIN {X 0,Y 316.958,Z 504.051,A -85,B 0,C 180,E1 -15588.252,E2 -15588.252} C_VEL
LIN {X 0,Y 318.169,Z 495.324,A -85,B 0,C 180,E1 -15589.349,E2 -15589.349} C_VEL
LIN {X 0,Y 318.614,Z 489.584,A -85,B 0,C 180,E1 -15589.992,E2 -15589.992} C_VEL
LIN {X 0,Y 317.51,Z 479.225,A -85,B 0,C 180,E1 -15591.073,E2 -15591.073} C_VEL
LIN {X 0,Y 316.107,Z 469.653,A -85,B 0,C 180,E1 -15591.923,E2 -15591.923} C_VEL
LIN {X 0,Y 314.062,Z 459.698,A -85,B 0,C 180,E1 -15592.684,E2 -15592.684} C_VEL
LIN {X 0,Y 311.33,Z 448.908,A -85,B 0,C 180,E1 -15593.369,E2 -15593.369} C_VEL
LIN {X 0,Y 311.246,Z 448.157,A -85,B 0,C 180,E1 -15593.432,E2 -15593.432} C_VEL
LIN {X 0,Y 311.577,Z 444.423,A -85,B 0,C 180,E1 -15596.815,E2 -15596.815} C_VEL
LIN {X 0,Y 312.22,Z 439.722,A -85,B 0,C 180,E1 -15601.198,E2 -15601.198} C_VEL
LIN {X 0,Y 312.59,Z 436.658,A -85,B 0,C 180,E1 -15604.199,E2 -15604.199} C_VEL
LIN {X 0,Y 313.038,Z 433.578,A -85,B 0,C 180,E1 -15607.312,E2 -15607.312} C_VEL
LIN {X 0,Y 313.475,Z 430.538,A -85,B 0,C 180,E1 -15610.553,E2 -15610.553} C_VEL
LIN {X 0,Y 313.564,Z 427.536,A -85,B 0,C 180,E1 -15614.011,E2 -15614.011} C_VEL
LIN {X 0,Y 313.301,Z 424.586,A -85,B 0,C 180,E1 -15617.703,E2 -15617.703} C_VEL
LIN {X 0,Y 312.95,Z 422.187,A -85,B 0,C 180,E1 -15621.037,E2 -15621.037} C_VEL
LIN {X 0,Y 312.666,Z 420.068,A -85,B 0,C 180,E1 -15624.237,E2 -15624.237} C_VEL
LIN {X 0,Y 312.518,Z 419.098,A -85,B 0,C 180,E1 -15625.791,E2 -15625.791} C_VEL
LIN {X 0,Y 312.525,Z 419.056,A -85,B 0,C 180,E1 -15628.853,E2 -15628.853} C_VEL
LIN {X 0,Y 312.571,Z 419.052,A -85,B 0,C 180,E1 -15631.824,E2 -15631.824} C_VEL
LIN {X 0,Y 312.581,Z 419.047,A -85,B 0,C 180,E1 -15634.71,E2 -15634.71} C_VEL
LIN {X 0,Y 312.532,Z 419.053,A -85,B 0,C 180,E1 -15638.912,E2 -15638.912} C_VEL
LIN {X 0,Y 312.633,Z 419.044,A -85,B 0,C 180,E1 -15641.655,E2 -15641.655} C_VEL
LIN {X 0,Y 312.688,Z 419.038,A -85,B 0,C 180,E1 -15645.685,E2 -15645.685} C_VEL
LIN {X 0,Y 312.692,Z 419.037,A -85,B 0,C 180,E1 -15649.641,E2 -15649.641} C_VEL
LIN {X 0,Y 312.847,Z 419.013,A -85,B 0,C 180,E1 -15652.253,E2 -15652.253} C_VEL
LIN {X 0,Y 312.71,Z 419.03,A -85,B 0,C 180,E1 -15654.842,E2 -15654.842} C_VEL
LIN {X 0,Y 312.984,Z 418.995,A -85,B 0,C 180,E1 -15658.713,E2 -15658.713} C_VEL
LIN {X 0,Y 312.984,Z 418.992,A -85,B 0,C 180,E1 -15661.286,E2 -15661.286} C_VEL
LIN {X 0,Y 312.71,Z 419.031,A -85,B 0,C 180,E1 -15665.157,E2 -15665.157} C_VEL
LIN {X 0,Y 312.846,Z 419.014,A -85,B 0,C 180,E1 -15667.746,E2 -15667.746} C_VEL
LIN {X 0,Y 312.661,Z 419.038,A -85,B 0,C 180,E1 -15671.671,E2 -15671.671} C_VEL
LIN {X 0,Y 312.693,Z 419.033,A -85,B 0,C 180,E1 -15674.887,E2 -15674.887} C_VEL
LIN {X 0,Y 312.623,Z 419.043,A -85,B 0,C 180,E1 -15679.236,E2 -15679.236} C_VEL
LIN {X 0,Y 312.538,Z 419.054,A -85,B 0,C 180,E1 -15682.789,E2 -15682.789} C_VEL
LIN {X 0,Y 312.595,Z 419.043,A -85,B 0,C 180,E1 -15685.935,E2 -15685.935} C_VEL
LIN {X 0,Y 312.538,Z 419.052,A -85,B 0,C 180,E1 -15689.65,E2 -15689.65} C_VEL
LIN {X 0,Y 312.512,Z 419.055,A -85,B 0,C 180,E1 -15693.689,E2 -15693.689} C_VEL
LIN {X 0,Y 312.534,Z 419.053,A -85,B 0,C 180,E1 -15697.383,E2 -15697.383} C_VEL
LIN {X 0,Y 312.519,Z 419.058,A -85,B 0,C 180,E1 -15700.704,E2 -15700.704} C_VEL
LIN {X 0,Y 312.523,Z 419.054,A -85,B 0,C 180,E1 -15704.196,E2 -15704.196} C_VEL
LIN {X 0,Y 312.481,Z 419.059,A -85,B 0,C 180,E1 -15707.918,E2 -15707.918} C_VEL
LIN {X 0,Y 312.529,Z 419.053,A -85,B 0,C 180,E1 -15711.91,E2 -15711.91} C_VEL
LIN {X 0,Y 312.501,Z 419.057,A -85,B 0,C 180,E1 -15715.79,E2 -15715.79} C_VEL
LIN {X 0,Y 312.515,Z 419.057,A -85,B 0,C 180,E1 -15718.854,E2 -15718.854} C_VEL
LIN {X 0,Y 312.565,Z 419.05,A -85,B 0,C 180,E1 -15721.825,E2 -15721.825} C_VEL
LIN {X 0,Y 312.58,Z 419.05,A -85,B 0,C 180,E1 -15724.711,E2 -15724.711} C_VEL
LIN {X 0,Y 312.55,Z 419.246,A -85,B 0,C 180,E1 -15726.366,E2 -15726.366} C_VEL
LIN {X 0,Y 313.724,Z 422.221,A -85,B 0,C 180,E1 -15726.547,E2 -15726.547} C_VEL
LIN {X 0,Y 316.617,Z 426.932,A -85,B 0,C 180,E1 -15726.949,E2 -15726.949} C_VEL
LIN {X 0,Y 319.708,Z 431.511,A -85,B 0,C 180,E1 -15727.406,E2 -15727.406} C_VEL
LIN {X 0,Y 323.565,Z 436.711,A -85,B 0,C 180,E1 -15728.039,E2 -15728.039} C_VEL
LIN {X 0,Y 328.119,Z 442.391,A -85,B 0,C 180,E1 -15728.844,E2 -15728.844} C_VEL
LIN {X 0,Y 332.62,Z 447.747,A -85,B 0,C 180,E1 -15729.703,E2 -15729.703} C_VEL
LIN {X 0,Y 338.087,Z 453.928,A -85,B 0,C 180,E1 -15730.841,E2 -15730.841} C_VEL
LIN {X 0,Y 343.829,Z 460.127,A -85,B 0,C 180,E1 -15732.146,E2 -15732.146} C_VEL
LIN {X 0,Y 349.866,Z 466.326,A -85,B 0,C 180,E1 -15733.667,E2 -15733.667} C_VEL
LIN {X 0,Y 352.528,Z 468.51,A -85,B 0,C 180,E1 -15734.346,E2 -15734.346} C_VEL
LIN {X 0,Y 356.93,Z 473.153,A -85,B 0,C 180,E1 -15735.674,E2 -15735.674} C_VEL
LIN {X 0,Y 361.432,Z 477.006,A -85,B 0,C 180,E1 -15737.111,E2 -15737.111} C_VEL
LIN {X 0,Y 365.572,Z 480.868,A -85,B 0,C 180,E1 -15738.65,E2 -15738.65} C_VEL
LIN {X 0,Y 369.376,Z 483.453,A -85,B 0,C 180,E1 -15740.14,E2 -15740.14} C_VEL
LIN {X 0,Y 371.589,Z 485.797,A -85,B 0,C 180,E1 -15741.298,E2 -15741.298} C_VEL
LIN {X 0,Y 373.464,Z 487.762,A -85,B 0,C 180,E1 -15742.431,E2 -15742.431} C_VEL
LIN {X 0,Y 375.25,Z 489.148,A -85,B 0,C 180,E1 -15743.548,E2 -15743.548} C_VEL
LIN {X 0,Y 376.772,Z 490.137,A -85,B 0,C 180,E1 -15744.649,E2 -15744.649} C_VEL
LIN {X 0,Y 378.092,Z 490.734,A -85,B 0,C 180,E1 -15745.736,E2 -15745.736} C_VEL
LIN {X 0,Y 379.829,Z 491.164,A -85,B 0,C 180,E1 -15747.641,E2 -15747.641} C_VEL
LIN {X 0,Y 380.477,Z 491.283,A -85,B 0,C 180,E1 -15748.942,E2 -15748.942} C_VEL
LIN {X 0,Y 380.635,Z 491.33,A -85,B 0,C 180,E1 -15750,E2 -15750} C_VEL
LIN {X 0,Y 380.474,Z 491.285,A -85,B 0,C 180,E1 -15751.058,E2 -15751.058} C_VEL
LIN {X 0,Y 379.822,Z 491.21,A -85,B 0,C 180,E1 -15752.332,E2 -15752.332} C_VEL
LIN {X 0,Y 378.084,Z 490.765,A -85,B 0,C 180,E1 -15754.264,E2 -15754.264} C_VEL
LIN {X 0,Y 376.798,Z 490.126,A -85,B 0,C 180,E1 -15755.351,E2 -15755.351} C_VEL
LIN {X 0,Y 374.979,Z 488.961,A -85,B 0,C 180,E1 -15756.62,E2 -15756.62} C_VEL
LIN {X 0,Y 373.503,Z 487.741,A -85,B 0,C 180,E1 -15757.569,E2 -15757.569} C_VEL
LIN {X 0,Y 370.365,Z 484.489,A -85,B 0,C 180,E1 -15759.344,E2 -15759.344} C_VEL
LIN {X 0,Y 369.381,Z 483.476,A -85,B 0,C 180,E1 -15759.86,E2 -15759.86} C_VEL
LIN {X 0,Y 365.565,Z 480.887,A -85,B 0,C 180,E1 -15761.344,E2 -15761.344} C_VEL
LIN {X 0,Y 361.944,Z 477.553,A -85,B 0,C 180,E1 -15762.696,E2 -15762.696} C_VEL
LIN {X 0,Y 358.275,Z 474.255,A -85,B 0,C 180,E1 -15763.909,E2 -15763.909} C_VEL
LIN {X 0,Y 353.799,Z 469.992,A -85,B 0,C 180,E1 -15765.26,E2 -15765.26} C_VEL
LIN {X 0,Y 347.938,Z 464.399,A -85,B 0,C 180,E1 -15766.838,E2 -15766.838} C_VEL
LIN {X 0,Y 340.823,Z 457.068,A -85,B 0,C 180,E1 -15768.545,E2 -15768.545} C_VEL
LIN {X 0,Y 337.511,Z 453.359,A -85,B 0,C 180,E1 -15769.283,E2 -15769.283} C_VEL
LIN {X 0,Y 330.252,Z 445.161,A -85,B 0,C 180,E1 -15770.743,E2 -15770.743} C_VEL
LIN {X 0,Y 324.324,Z 437.662,A -85,B 0,C 180,E1 -15771.832,E2 -15771.832} C_VEL
LIN {X 0,Y 320.427,Z 432.582,A -85,B 0,C 180,E1 -15772.477,E2 -15772.477} C_VEL
LIN {X 0,Y 317.061,Z 427.615,A -85,B 0,C 180,E1 -15772.988,E2 -15772.988} C_VEL
LIN {X 0,Y 314.598,Z 423.676,A -85,B 0,C 180,E1 -15773.338,E2 -15773.338} C_VEL
LIN {X 0,Y 312.73,Z 420.098,A -85,B 0,C 180,E1 -15773.595,E2 -15773.595} C_VEL
LIN {X 0,Y 312.534,Z 419.057,A -85,B 0,C 180,E1 -15773.666,E2 -15773.666} C_VEL
LIN {X 0,Y 312.547,Z 419.051,A -85,B 0,C 180,E1 -15776.725,E2 -15776.725} C_VEL
LIN {X 0,Y 312.533,Z 419.057,A -85,B 0,C 180,E1 -15779.651,E2 -15779.651} C_VEL
LIN {X 0,Y 312.514,Z 419.058,A -85,B 0,C 180,E1 -15783.689,E2 -15783.689} C_VEL
LIN {X 0,Y 312.532,Z 419.057,A -85,B 0,C 180,E1 -15787.383,E2 -15787.383} C_VEL
LIN {X 0,Y 312.484,Z 419.059,A -85,B 0,C 180,E1 -15790.709,E2 -15790.709} C_VEL
LIN {X 0,Y 312.466,Z 419.06,A -85,B 0,C 180,E1 -15794.206,E2 -15794.206} C_VEL
LIN {X 0,Y 312.479,Z 419.059,A -85,B 0,C 180,E1 -15797.918,E2 -15797.918} C_VEL
LIN {X 0,Y 312.491,Z 419.061,A -85,B 0,C 180,E1 -15800.971,E2 -15800.971} C_VEL
LIN {X 0,Y 312.525,Z 419.052,A -85,B 0,C 180,E1 -15804.22,E2 -15804.22} C_VEL
LIN {X 0,Y 312.497,Z 419.059,A -85,B 0,C 180,E1 -15807.334,E2 -15807.334} C_VEL
LIN {X 0,Y 312.545,Z 419.053,A -85,B 0,C 180,E1 -15811.276,E2 -15811.276} C_VEL
LIN {X 0,Y 312.578,Z 419.049,A -85,B 0,C 180,E1 -15814.711,E2 -15814.711} C_VEL
LIN {X 0,Y 312.58,Z 419.047,A -85,B 0,C 180,E1 -15817.529,E2 -15817.529} C_VEL
LIN {X 0,Y 312.631,Z 419.04,A -85,B 0,C 180,E1 -15821.657,E2 -15821.657} C_VEL
LIN {X 0,Y 312.686,Z 419.031,A -85,B 0,C 180,E1 -15825.687,E2 -15825.687} C_VEL
LIN {X 0,Y 312.691,Z 419.031,A -85,B 0,C 180,E1 -15829.642,E2 -15829.642} C_VEL
LIN {X 0,Y 312.846,Z 419.014,A -85,B 0,C 180,E1 -15832.254,E2 -15832.254} C_VEL
LIN {X 0,Y 312.71,Z 419.031,A -85,B 0,C 180,E1 -15834.843,E2 -15834.843} C_VEL
LIN {X 0,Y 312.716,Z 419.026,A -85,B 0,C 180,E1 -15836.335,E2 -15836.335} C_VEL
LIN {X 0,Y 312.185,Z 419.088,A -85,B 0,C 180,E1 -15837.414,E2 -15837.414} C_VEL
LIN {X 0,Y 309.451,Z 419.431,A -85,B 0,C 180,E1 -15839.171,E2 -15839.171} C_VEL
LIN {X 0,Y 307.046,Z 419.736,A -85,B 0,C 180,E1 -15840.597,E2 -15840.597} C_VEL
LIN {X 0,Y 305.987,Z 419.866,A -85,B 0,C 180,E1 -15841.699,E2 -15841.699} C_VEL
LIN {X 0,Y 305.89,Z 419.879,A -85,B 0,C 180,E1 -15842.072,E2 -15842.072} C_VEL
LIN {X 0,Y 305.836,Z 419.89,A -85,B 0,C 180,E1 -15846.598,E2 -15846.598} C_VEL
LIN {X 0,Y 305.698,Z 419.904,A -85,B 0,C 180,E1 -15849.262,E2 -15849.262} C_VEL
LIN {X 0,Y 305.583,Z 419.918,A -85,B 0,C 180,E1 -15853.297,E2 -15853.297} C_VEL
LIN {X 0,Y 305.589,Z 419.921,A -85,B 0,C 180,E1 -15856.021,E2 -15856.021} C_VEL
LIN {X 0,Y 305.555,Z 419.922,A -85,B 0,C 180,E1 -15859.437,E2 -15859.437} C_VEL
LIN {X 0,Y 305.482,Z 419.932,A -85,B 0,C 180,E1 -15863.04,E2 -15863.04} C_VEL
LIN {X 0,Y 305.544,Z 419.928,A -85,B 0,C 180,E1 -15866.228,E2 -15866.228} C_VEL
LIN {X 0,Y 305.493,Z 419.93,A -85,B 0,C 180,E1 -15869.051,E2 -15869.051} C_VEL
LIN {X 0,Y 305.445,Z 419.941,A -85,B 0,C 180,E1 -15871.953,E2 -15871.953} C_VEL
LIN {X 0,Y 305.507,Z 420.145,A -85,B 0,C 180,E1 -15874.092,E2 -15874.092} C_VEL
LIN {X 0,Y 305.863,Z 422.838,A -85,B 0,C 180,E1 -15878.346,E2 -15878.346} C_VEL
LIN {X 0,Y 306.226,Z 425.205,A -85,B 0,C 180,E1 -15881.726,E2 -15881.726} C_VEL
LIN {X 0,Y 306.502,Z 427.948,A -85,B 0,C 180,E1 -15885.303,E2 -15885.303} C_VEL
LIN {X 0,Y 306.465,Z 430.46,A -85,B 0,C 180,E1 -15888.316,E2 -15888.316} C_VEL
LIN {X 0,Y 306.104,Z 433.492,A -85,B 0,C 180,E1 -15891.692,E2 -15891.692} C_VEL
LIN {X 0,Y 305.643,Z 436.544,A -85,B 0,C 180,E1 -15894.912,E2 -15894.912} C_VEL
LIN {X 0,Y 305.184,Z 440.03,A -85,B 0,C 180,E1 -15898.438,E2 -15898.438} C_VEL
LIN {X 0,Y 304.563,Z 444.273,A -85,B 0,C 180,E1 -15902.516,E2 -15902.516} C_VEL
LIN {X 0,Y 304.227,Z 447.999,A -85,B 0,C 180,E1 -15906.008,E2 -15906.008} C_VEL
LIN {X 0,Y 307.765,Z 462.363,A -85,B 0,C 180,E1 -15906.973,E2 -15906.973} C_VEL
LIN {X 0,Y 310.051,Z 474.808,A -85,B 0,C 180,E1 -15908.032,E2 -15908.032} C_VEL
LIN {X 0,Y 311.272,Z 484.453,A -85,B 0,C 180,E1 -15908.997,E2 -15908.997} C_VEL
LIN {X 0,Y 311.868,Z 492.424,A -85,B 0,C 180,E1 -15909.9,E2 -15909.9} C_VEL
LIN {X 0,Y 310.377,Z 502.719,A -85,B 0,C 180,E1 -15911.176,E2 -15911.176} C_VEL
LIN {X 0,Y 309.107,Z 511.249,A -85,B 0,C 180,E1 -15912.467,E2 -15912.467} C_VEL
LIN {X 0,Y 307.978,Z 519.024,A -85,B 0,C 180,E1 -15913.883,E2 -15913.883} C_VEL
LIN {X 0,Y 306.841,Z 526.048,A -85,B 0,C 180,E1 -15915.408,E2 -15915.408} C_VEL
LIN {X 0,Y 305.755,Z 532.363,A -85,B 0,C 180,E1 -15917.05,E2 -15917.05} C_VEL
LIN {X 0,Y 304.981,Z 537.627,A -85,B 0,C 180,E1 -15918.704,E2 -15918.704} C_VEL
LIN {X 0,Y 304.31,Z 542.759,A -85,B 0,C 180,E1 -15920.697,E2 -15920.697} C_VEL
LIN {X 0,Y 303.844,Z 546.748,A -85,B 0,C 180,E1 -15922.691,E2 -15922.691} C_VEL
LIN {X 0,Y 303.62,Z 549.699,A -85,B 0,C 180,E1 -15924.688,E2 -15924.688} C_VEL
LIN {X 0,Y 303.608,Z 552.15,A -85,B 0,C 180,E1 -15927.347,E2 -15927.347} C_VEL
LIN {X 0,Y 303.567,Z 552.739,A -85,B 0,C 180,E1 -15928.673,E2 -15928.673} C_VEL
LIN {X 0,Y 303.567,Z 552.739,A -85,B 0,C 180,E1 -15931.327,E2 -15931.327} C_VEL
LIN {X 0,Y 303.608,Z 552.15,A -85,B 0,C 180,E1 -15932.653,E2 -15932.653} C_VEL
LIN {X 0,Y 303.64,Z 549.7,A -85,B 0,C 180,E1 -15935.312,E2 -15935.312} C_VEL
LIN {X 0,Y 303.844,Z 546.748,A -85,B 0,C 180,E1 -15937.309,E2 -15937.309} C_VEL
LIN {X 0,Y 304.31,Z 542.759,A -85,B 0,C 180,E1 -15939.303,E2 -15939.303} C_VEL
LIN {X 0,Y 304.981,Z 537.627,A -85,B 0,C 180,E1 -15941.296,E2 -15941.296} C_VEL
LIN {X 0,Y 305.755,Z 532.363,A -85,B 0,C 180,E1 -15942.95,E2 -15942.95} C_VEL
LIN {X 0,Y 306.846,Z 526.048,A -85,B 0,C 180,E1 -15944.592,E2 -15944.592} C_VEL
LIN {X 0,Y 307.772,Z 520.096,A -85,B 0,C 180,E1 -15945.903,E2 -15945.903} C_VEL
LIN {X 0,Y 308.755,Z 513.166,A -85,B 0,C 180,E1 -15947.212,E2 -15947.212} C_VEL
LIN {X 0,Y 310.024,Z 504.987,A -85,B 0,C 180,E1 -15948.503,E2 -15948.503} C_VEL
LIN {X 0,Y 311.285,Z 496.478,A -85,B 0,C 180,E1 -15949.623,E2 -15949.623} C_VEL
LIN {X 0,Y 311.836,Z 490.999,A -85,B 0,C 180,E1 -15950.274,E2 -15950.274} C_VEL
LIN {X 0,Y 310.621,Z 479.032,A -85,B 0,C 180,E1 -15951.562,E2 -15951.562} C_VEL
LIN {X 0,Y 309.287,Z 469.97,A -85,B 0,C 180,E1 -15952.397,E2 -15952.397} C_VEL
LIN {X 0,Y 306.972,Z 458.876,A -85,B 0,C 180,E1 -15953.269,E2 -15953.269} C_VEL
LIN {X 0,Y 304.262,Z 448.63,A -85,B 0,C 180,E1 -15953.948,E2 -15953.948} C_VEL
LIN {X 0,Y 304.212,Z 447.987,A -85,B 0,C 180,E1 -15954.005,E2 -15954.005} C_VEL
LIN {X 0,Y 304.558,Z 444.252,A -85,B 0,C 180,E1 -15957.485,E2 -15957.485} C_VEL
LIN {X 0,Y 305.185,Z 440.03,A -85,B 0,C 180,E1 -15961.562,E2 -15961.562} C_VEL
LIN {X 0,Y 305.625,Z 436.526,A -85,B 0,C 180,E1 -15965.091,E2 -15965.091} C_VEL
LIN {X 0,Y 306.166,Z 433.099,A -85,B 0,C 180,E1 -15968.696,E2 -15968.696} C_VEL
LIN {X 0,Y 306.464,Z 430.439,A -85,B 0,C 180,E1 -15971.685,E2 -15971.685} C_VEL
LIN {X 0,Y 306.459,Z 427.45,A -85,B 0,C 180,E1 -15975.308,E2 -15975.308} C_VEL
LIN {X 0,Y 306.132,Z 424.488,A -85,B 0,C 180,E1 -15979.251,E2 -15979.251} C_VEL
LIN {X 0,Y 305.703,Z 421.774,A -85,B 0,C 180,E1 -15983.292,E2 -15983.292} C_VEL
LIN {X 0,Y 305.467,Z 419.94,A -85,B 0,C 180,E1 -15986.483,E2 -15986.483} C_VEL
LIN {X 0,Y 305.463,Z 419.938,A -85,B 0,C 180,E1 -15989.59,E2 -15989.59} C_VEL
LIN {X 0,Y 305.518,Z 419.927,A -85,B 0,C 180,E1 -15992.608,E2 -15992.608} C_VEL
LIN {X 0,Y 305.5,Z 419.931,A -85,B 0,C 180,E1 -15995.537,E2 -15995.537} C_VEL
LIN {X 0,Y 305.502,Z 419.933,A -85,B 0,C 180,E1 -15999.813,E2 -15999.813} C_VEL
LIN {X 0,Y 305.569,Z 419.92,A -85,B 0,C 180,E1 -16002.602,E2 -16002.602} C_VEL
LIN {X 0,Y 305.644,Z 419.913,A -85,B 0,C 180,E1 -16005.348,E2 -16005.348} C_VEL
LIN {X 0,Y 305.629,Z 419.915,A -85,B 0,C 180,E1 -16009.399,E2 -16009.399} C_VEL
LIN {X 0,Y 305.791,Z 419.893,A -85,B 0,C 180,E1 -16012.073,E2 -16012.073} C_VEL
LIN {X 0,Y 305.681,Z 419.905,A -85,B 0,C 180,E1 -16014.723,E2 -16014.723} C_VEL
LIN {X 0,Y 305.95,Z 419.871,A -85,B 0,C 180,E1 -16018.683,E2 -16018.683} C_VEL
LIN {X 0,Y 305.95,Z 419.867,A -85,B 0,C 180,E1 -16021.316,E2 -16021.316} C_VEL
LIN {X 0,Y 305.681,Z 419.907,A -85,B 0,C 180,E1 -16025.276,E2 -16025.276} C_VEL
LIN {X 0,Y 305.79,Z 419.892,A -85,B 0,C 180,E1 -16027.926,E2 -16027.926} C_VEL
LIN {X 0,Y 305.595,Z 419.917,A -85,B 0,C 180,E1 -16031.945,E2 -16031.945} C_VEL
LIN {X 0,Y 305.631,Z 419.913,A -85,B 0,C 180,E1 -16035.034,E2 -16035.034} C_VEL
LIN {X 0,Y 305.57,Z 419.92,A -85,B 0,C 180,E1 -16039.444,E2 -16039.444} C_VEL
LIN {X 0,Y 305.483,Z 419.935,A -85,B 0,C 180,E1 -16043.041,E2 -16043.041} C_VEL
LIN {X 0,Y 305.54,Z 419.922,A -85,B 0,C 180,E1 -16046.227,E2 -16046.227} C_VEL
LIN {X 0,Y 305.489,Z 419.934,A -85,B 0,C 180,E1 -16049.05,E2 -16049.05} C_VEL
LIN {X 0,Y 305.458,Z 419.934,A -85,B 0,C 180,E1 -16053.517,E2 -16053.517} C_VEL
LIN {X 0,Y 305.49,Z 419.933,A -85,B 0,C 180,E1 -16056.736,E2 -16056.736} C_VEL
LIN {X 0,Y 305.478,Z 419.934,A -85,B 0,C 180,E1 -16060.606,E2 -16060.606} C_VEL
LIN {X 0,Y 305.484,Z 419.93,A -85,B 0,C 180,E1 -16063.644,E2 -16063.644} C_VEL
LIN {X 0,Y 305.457,Z 419.934,A -85,B 0,C 180,E1 -16067.413,E2 -16067.413} C_VEL
LIN {X 0,Y 305.489,Z 419.93,A -85,B 0,C 180,E1 -16071.601,E2 -16071.601} C_VEL
LIN {X 0,Y 305.457,Z 419.937,A -85,B 0,C 180,E1 -16074.887,E2 -16074.887} C_VEL
LIN {X 0,Y 305.444,Z 419.94,A -85,B 0,C 180,E1 -16078.356,E2 -16078.356} C_VEL
LIN {X 0,Y 305.508,Z 419.929,A -85,B 0,C 180,E1 -16081.113,E2 -16081.113} C_VEL
LIN {X 0,Y 305.566,Z 419.924,A -85,B 0,C 180,E1 -16084.088,E2 -16084.088} C_VEL
LIN {X 0,Y 305.497,Z 419.931,A -85,B 0,C 180,E1 -16085.749,E2 -16085.749} C_VEL
LIN {X 0,Y 306.515,Z 422.773,A -85,B 0,C 180,E1 -16085.926,E2 -16085.926} C_VEL
LIN {X 0,Y 310.716,Z 430.413,A -85,B 0,C 180,E1 -16086.487,E2 -16086.487} C_VEL
LIN {X 0,Y 316.495,Z 438.83,A -85,B 0,C 180,E1 -16087.355,E2 -16087.355} C_VEL
LIN {X 0,Y 323.302,Z 447.316,A -85,B 0,C 180,E1 -16088.517,E2 -16088.517} C_VEL
LIN {X 0,Y 328.316,Z 453.236,A -85,B 0,C 180,E1 -16089.473,E2 -16089.473} C_VEL
LIN {X 0,Y 333.438,Z 459.106,A -85,B 0,C 180,E1 -16090.549,E2 -16090.549} C_VEL
LIN {X 0,Y 339.91,Z 465.994,A -85,B 0,C 180,E1 -16092.005,E2 -16092.005} C_VEL
LIN {X 0,Y 345.627,Z 471.866,A -85,B 0,C 180,E1 -16093.461,E2 -16093.461} C_VEL
LIN {X 0,Y 349.866,Z 475.86,A -85,B 0,C 180,E1 -16094.621,E2 -16094.621} C_VEL
LIN {X 0,Y 352.763,Z 478.806,A -85,B 0,C 180,E1 -16095.501,E2 -16095.501} C_VEL
LIN {X 0,Y 357.214,Z 482.598,A -85,B 0,C 180,E1 -16096.908,E2 -16096.908} C_VEL
LIN {X 0,Y 361.423,Z 486.585,A -85,B 0,C 180,E1 -16098.469,E2 -16098.469} C_VEL
LIN {X 0,Y 365.471,Z 489.381,A -85,B 0,C 180,E1 -16100.034,E2 -16100.034} C_VEL
LIN {X 0,Y 369.042,Z 493.098,A -85,B 0,C 180,E1 -16102,E2 -16102} C_VEL
LIN {X 0,Y 371.384,Z 495.085,A -85,B 0,C 180,E1 -16103.481,E2 -16103.481} C_VEL
LIN {X 0,Y 373.764,Z 496.498,A -85,B 0,C 180,E1 -16105.247,E2 -16105.247} C_VEL
LIN {X 0,Y 375.389,Z 497.043,A -85,B 0,C 180,E1 -16106.78,E2 -16106.78} C_VEL
LIN {X 0,Y 376.24,Z 497.212,A -85,B 0,C 180,E1 -16107.859,E2 -16107.859} C_VEL
LIN {X 0,Y 376.751,Z 497.32,A -85,B 0,C 180,E1 -16108.931,E2 -16108.931} C_VEL
LIN {X 0,Y 376.918,Z 497.366,A -85,B 0,C 180,E1 -16110,E2 -16110} C_VEL
LIN {X 0,Y 376.749,Z 497.32,A -85,B 0,C 180,E1 -16111.069,E2 -16111.069} C_VEL
LIN {X 0,Y 376.207,Z 497.254,A -85,B 0,C 180,E1 -16112.141,E2 -16112.141} C_VEL
LIN {X 0,Y 375.389,Z 497.03,A -85,B 0,C 180,E1 -16113.22,E2 -16113.22} C_VEL
LIN {X 0,Y 373.76,Z 496.513,A -85,B 0,C 180,E1 -16114.745,E2 -16114.745} C_VEL
LIN {X 0,Y 371.367,Z 495.076,A -85,B 0,C 180,E1 -16116.52,E2 -16116.52} C_VEL
LIN {X 0,Y 369.051,Z 493.066,A -85,B 0,C 180,E1 -16118.009,E2 -16118.009} C_VEL
LIN {X 0,Y 365.473,Z 489.39,A -85,B 0,C 180,E1 -16119.966,E2 -16119.966} C_VEL
LIN {X 0,Y 361.416,Z 486.578,A -85,B 0,C 180,E1 -16121.533,E2 -16121.533} C_VEL
LIN {X 0,Y 357.186,Z 482.597,A -85,B 0,C 180,E1 -16123.094,E2 -16123.094} C_VEL
LIN {X 0,Y 352.735,Z 478.764,A -85,B 0,C 180,E1 -16124.501,E2 -16124.501} C_VEL
LIN {X 0,Y 346.847,Z 472.931,A -85,B 0,C 180,E1 -16126.232,E2 -16126.232} C_VEL
LIN {X 0,Y 340.917,Z 466.928,A -85,B 0,C 180,E1 -16127.758,E2 -16127.758} C_VEL
LIN {X 0,Y 335.295,Z 461.078,A -85,B 0,C 180,E1 -16129.05,E2 -16129.05} C_VEL
LIN {X 0,Y 329.626,Z 454.781,A -85,B 0,C 180,E1 -16130.263,E2 -16130.263} C_VEL
LIN {X 0,Y 323.885,Z 447.98,A -85,B 0,C 180,E1 -16131.374,E2 -16131.374} C_VEL
LIN {X 0,Y 319.399,Z 442.402,A -85,B 0,C 180,E1 -16132.177,E2 -16132.177} C_VEL
LIN {X 0,Y 315.29,Z 437.014,A -85,B 0,C 180,E1 -16132.844,E2 -16132.844} C_VEL
LIN {X 0,Y 310.112,Z 429.489,A -85,B 0,C 180,E1 -16133.595,E2 -16133.595} C_VEL
LIN {X 0,Y 305.907,Z 421.572,A -85,B 0,C 180,E1 -16134.155,E2 -16134.155} C_VEL
LIN {X 0,Y 305.491,Z 419.932,A -85,B 0,C 180,E1 -16134.268,E2 -16134.268} C_VEL
LIN {X 0,Y 305.513,Z 419.931,A -85,B 0,C 180,E1 -16137.391,E2 -16137.391} C_VEL
LIN {X 0,Y 305.452,Z 419.935,A -85,B 0,C 180,E1 -16140.409,E2 -16140.409} C_VEL
LIN {X 0,Y 305.459,Z 419.934,A -85,B 0,C 180,E1 -16144.078,E2 -16144.078} C_VEL
LIN {X 0,Y 305.49,Z 419.93,A -85,B 0,C 180,E1 -16146.736,E2 -16146.736} C_VEL
LIN {X 0,Y 305.449,Z 419.935,A -85,B 0,C 180,E1 -16150.6,E2 -16150.6} C_VEL
LIN {X 0,Y 305.412,Z 419.939,A -85,B 0,C 180,E1 -16154.492,E2 -16154.492} C_VEL
LIN {X 0,Y 305.435,Z 419.936,A -85,B 0,C 180,E1 -16158.143,E2 -16158.143} C_VEL
LIN {X 0,Y 305.46,Z 419.935,A -85,B 0,C 180,E1 -16161.596,E2 -16161.596} C_VEL
LIN {X 0,Y 305.455,Z 419.936,A -85,B 0,C 180,E1 -16164.887,E2 -16164.887} C_VEL
LIN {X 0,Y 305.444,Z 419.936,A -85,B 0,C 180,E1 -16168.355,E2 -16168.355} C_VEL
LIN {X 0,Y 305.514,Z 419.93,A -85,B 0,C 180,E1 -16171.114,E2 -16171.114} C_VEL
LIN {X 0,Y 305.564,Z 419.919,A -85,B 0,C 180,E1 -16174.088,E2 -16174.088} C_VEL
LIN {X 0,Y 305.494,Z 419.93,A -85,B 0,C 180,E1 -16178.403,E2 -16178.403} C_VEL
LIN {X 0,Y 305.583,Z 419.92,A -85,B 0,C 180,E1 -16181.218,E2 -16181.218} C_VEL
LIN {X 0,Y 305.641,Z 419.91,A -85,B 0,C 180,E1 -16185.349,E2 -16185.349} C_VEL
LIN {X 0,Y 305.628,Z 419.911,A -85,B 0,C 180,E1 -16189.4,E2 -16189.4} C_VEL
LIN {X 0,Y 305.79,Z 419.892,A -85,B 0,C 180,E1 -16192.074,E2 -16192.074} C_VEL
LIN {X 0,Y 305.681,Z 419.907,A -85,B 0,C 180,E1 -16194.724,E2 -16194.724} C_VEL
LIN {X 0,Y 305.95,Z 419.867,A -85,B 0,C 180,E1 -16198.684,E2 -16198.684} C_VEL
LIN {X 0,Y 305.95,Z 419.871,A -85,B 0,C 180,E1 -16201.317,E2 -16201.317} C_VEL
LIN {X 0,Y 305.89,Z 419.879,A -85,B 0,C 180,E1 -16202.072,E2 -16202.072} C_VEL
LIN {X 0,Y 305.185,Z 419.97,A -85,B 0,C 180,E1 -16203.17,E2 -16203.17} C_VEL
LIN {X 0,Y 302.282,Z 420.33,A -85,B 0,C 180,E1 -16204.955,E2 -16204.955} C_VEL
LIN {X 0,Y 299.844,Z 420.637,A -85,B 0,C 180,E1 -16206.403,E2 -16206.403} C_VEL
LIN {X 0,Y 298.81,Z 420.762,A -85,B 0,C 180,E1 -16207.525,E2 -16207.525} C_VEL
LIN {X 0,Y 298.731,Z 420.773,A -85,B 0,C 180,E1 -16207.905,E2 -16207.905} C_VEL
LIN {X 0,Y 298.548,Z 420.799,A -85,B 0,C 180,E1 -16212.232,E2 -16212.232} C_VEL
LIN {X 0,Y 298.58,Z 420.791,A -85,B 0,C 180,E1 -16215.195,E2 -16215.195} C_VEL
LIN {X 0,Y 298.521,Z 420.798,A -85,B 0,C 180,E1 -16219.245,E2 -16219.245} C_VEL
LIN {X 0,Y 298.425,Z 420.812,A -85,B 0,C 180,E1 -16223.601,E2 -16223.601} C_VEL
LIN {X 0,Y 298.486,Z 420.805,A -85,B 0,C 180,E1 -16226.575,E2 -16226.575} C_VEL
LIN {X 0,Y 298.419,Z 420.814,A -85,B 0,C 180,E1 -16229.642,E2 -16229.642} C_VEL
LIN {X 0,Y 298.396,Z 420.819,A -85,B 0,C 180,E1 -16232.801,E2 -16232.801} C_VEL
LIN {X 0,Y 298.527,Z 421.516,A -85,B 0,C 180,E1 -16234.517,E2 -16234.517} C_VEL
LIN {X 0,Y 298.774,Z 423.5,A -85,B 0,C 180,E1 -16237.706,E2 -16237.706} C_VEL
LIN {X 0,Y 299.143,Z 425.881,A -85,B 0,C 180,E1 -16241.255,E2 -16241.255} C_VEL
LIN {X 0,Y 299.455,Z 428.477,A -85,B 0,C 180,E1 -16244.756,E2 -16244.756} C_VEL
LIN {X 0,Y 299.483,Z 430.362,A -85,B 0,C 180,E1 -16247.115,E2 -16247.115} C_VEL
LIN {X 0,Y 299.394,Z 431.859,A -85,B 0,C 180,E1 -16248.909,E2 -16248.909} C_VEL
LIN {X 0,Y 298.934,Z 434.882,A -85,B 0,C 180,E1 -16252.32,E2 -16252.32} C_VEL
LIN {X 0,Y 298.508,Z 437.942,A -85,B 0,C 180,E1 -16255.595,E2 -16255.595} C_VEL
LIN {X 0,Y 298.056,Z 441.025,A -85,B 0,C 180,E1 -16258.752,E2 -16258.752} C_VEL
LIN {X 0,Y 297.405,Z 445.66,A -85,B 0,C 180,E1 -16263.322,E2 -16263.322} C_VEL
LIN {X 0,Y 297.196,Z 448.037,A -85,B 0,C 180,E1 -16265.432,E2 -16265.432} C_VEL
LIN {X 0,Y 299.856,Z 458.352,A -85,B 0,C 180,E1 -16266.128,E2 -16266.128} C_VEL
LIN {X 0,Y 301.916,Z 467.305,A -85,B 0,C 180,E1 -16266.854,E2 -16266.854} C_VEL
LIN {X 0,Y 303.494,Z 477.165,A -85,B 0,C 180,E1 -16267.758,E2 -16267.758} C_VEL
LIN {X 0,Y 304.526,Z 485.89,A -85,B 0,C 180,E1 -16268.686,E2 -16268.686} C_VEL
LIN {X 0,Y 305.023,Z 493.579,A -85,B 0,C 180,E1 -16269.605,E2 -16269.605} C_VEL
LIN {X 0,Y 303.668,Z 502.522,A -85,B 0,C 180,E1 -16270.744,E2 -16270.744} C_VEL
LIN {X 0,Y 302.323,Z 511.051,A -85,B 0,C 180,E1 -16272.061,E2 -16272.061} C_VEL
LIN {X 0,Y 301.205,Z 518.429,A -85,B 0,C 180,E1 -16273.426,E2 -16273.426} C_VEL
LIN {X 0,Y 300.164,Z 524.474,A -85,B 0,C 180,E1 -16274.728,E2 -16274.728} C_VEL
LIN {X 0,Y 299.032,Z 531.01,A -85,B 0,C 180,E1 -16276.407,E2 -16276.407} C_VEL
LIN {X 0,Y 298.249,Z 535.511,A -85,B 0,C 180,E1 -16277.756,E2 -16277.756} C_VEL
LIN {X 0,Y 297.469,Z 541.006,A -85,B 0,C 180,E1 -16279.794,E2 -16279.794} C_VEL
LIN {X 0,Y 296.929,Z 545.333,A -85,B 0,C 180,E1 -16281.836,E2 -16281.836} C_VEL
LIN {X 0,Y 296.689,Z 547.701,A -85,B 0,C 180,E1 -16283.198,E2 -16283.198} C_VEL
LIN {X 0,Y 296.528,Z 550.893,A -85,B 0,C 180,E1 -16285.923,E2 -16285.923} C_VEL
LIN {X 0,Y 296.535,Z 551.954,A -85,B 0,C 180,E1 -16287.283,E2 -16287.283} C_VEL
LIN {X 0,Y 296.487,Z 552.542,A -85,B 0,C 180,E1 -16288.642,E2 -16288.642} C_VEL
LIN {X 0,Y 296.487,Z 552.542,A -85,B 0,C 180,E1 -16291.358,E2 -16291.358} C_VEL
LIN {X 0,Y 296.535,Z 551.954,A -85,B 0,C 180,E1 -16292.717,E2 -16292.717} C_VEL
LIN {X 0,Y 296.549,Z 549.411,A -85,B 0,C 180,E1 -16295.508,E2 -16295.508} C_VEL
LIN {X 0,Y 296.797,Z 546.551,A -85,B 0,C 180,E1 -16297.483,E2 -16297.483} C_VEL
LIN {X 0,Y 297.277,Z 542.561,A -85,B 0,C 180,E1 -16299.525,E2 -16299.525} C_VEL
LIN {X 0,Y 297.972,Z 537.428,A -85,B 0,C 180,E1 -16301.565,E2 -16301.565} C_VEL
LIN {X 0,Y 298.82,Z 532.166,A -85,B 0,C 180,E1 -16303.256,E2 -16303.256} C_VEL
LIN {X 0,Y 299.943,Z 525.85,A -85,B 0,C 180,E1 -16304.936,E2 -16304.936} C_VEL
LIN {X 0,Y 300.938,Z 519.899,A -85,B 0,C 180,E1 -16306.274,E2 -16306.274} C_VEL
LIN {X 0,Y 301.961,Z 512.969,A -85,B 0,C 180,E1 -16307.612,E2 -16307.612} C_VEL
LIN {X 0,Y 303.29,Z 504.79,A -85,B 0,C 180,E1 -16308.93,E2 -16308.93} C_VEL
LIN {X 0,Y 304.603,Z 496.281,A -85,B 0,C 180,E1 -16310.072,E2 -16310.072} C_VEL
LIN {X 0,Y 305.026,Z 492.222,A -85,B 0,C 180,E1 -16310.571,E2 -16310.571} C_VEL
LIN {X 0,Y 303.808,Z 479.353,A -85,B 0,C 180,E1 -16312.024,E2 -16312.024} C_VEL
LIN {X 0,Y 302.151,Z 468.573,A -85,B 0,C 180,E1 -16313.039,E2 -16313.039} C_VEL
LIN {X 0,Y 299.854,Z 458.369,A -85,B 0,C 180,E1 -16313.871,E2 -16313.871} C_VEL
LIN {X 0,Y 297.188,Z 447.818,A -85,B 0,C 180,E1 -16314.604,E2 -16314.604} C_VEL
LIN {X 0,Y 297.576,Z 444.099,A -85,B 0,C 180,E1 -16318.186,E2 -16318.186} C_VEL
LIN {X 0,Y 298.144,Z 440.32,A -85,B 0,C 180,E1 -16321.938,E2 -16321.938} C_VEL
LIN {X 0,Y 298.697,Z 436.394,A -85,B 0,C 180,E1 -16326.03,E2 -16326.03} C_VEL
LIN {X 0,Y 299.186,Z 433.335,A -85,B 0,C 180,E1 -16329.363,E2 -16329.363} C_VEL
LIN {X 0,Y 299.399,Z 431.652,A -85,B 0,C 180,E1 -16331.308,E2 -16331.308} C_VEL
LIN {X 0,Y 299.457,Z 428.832,A -85,B 0,C 180,E1 -16334.753,E2 -16334.753} C_VEL
LIN {X 0,Y 299.152,Z 425.88,A -85,B 0,C 180,E1 -16338.743,E2 -16338.743} C_VEL
LIN {X 0,Y 298.771,Z 423.477,A -85,B 0,C 180,E1 -16342.294,E2 -16342.294} C_VEL
LIN {X 0,Y 298.505,Z 421.457,A -85,B 0,C 180,E1 -16345.593,E2 -16345.593} C_VEL
LIN {X 0,Y 298.396,Z 420.821,A -85,B 0,C 180,E1 -16347.199,E2 -16347.199} C_VEL
LIN {X 0,Y 298.429,Z 420.812,A -85,B 0,C 180,E1 -16350.613,E2 -16350.613} C_VEL
LIN {X 0,Y 298.48,Z 420.805,A -85,B 0,C 180,E1 -16353.473,E2 -16353.473} C_VEL
LIN {X 0,Y 298.427,Z 420.81,A -85,B 0,C 180,E1 -16356.698,E2 -16356.698} C_VEL
LIN {X 0,Y 298.521,Z 420.798,A -85,B 0,C 180,E1 -16360.755,E2 -16360.755} C_VEL
LIN {X 0,Y 298.588,Z 420.79,A -85,B 0,C 180,E1 -16364.994,E2 -16364.994} C_VEL
LIN {X 0,Y 298.586,Z 420.791,A -85,B 0,C 180,E1 -16369.146,E2 -16369.146} C_VEL
LIN {X 0,Y 298.735,Z 420.773,A -85,B 0,C 180,E1 -16371.885,E2 -16371.885} C_VEL
LIN {X 0,Y 298.652,Z 420.781,A -85,B 0,C 180,E1 -16374.598,E2 -16374.598} C_VEL
LIN {X 0,Y 298.917,Z 420.747,A -85,B 0,C 180,E1 -16378.652,E2 -16378.652} C_VEL
LIN {X 0,Y 298.917,Z 420.741,A -85,B 0,C 180,E1 -16381.346,E2 -16381.346} C_VEL
LIN {X 0,Y 298.781,Z 420.766,A -85,B 0,C 180,E1 -16386.753,E2 -16386.753} C_VEL
LIN {X 0,Y 298.628,Z 420.786,A -85,B 0,C 180,E1 -16389.481,E2 -16389.481} C_VEL
LIN {X 0,Y 298.545,Z 420.795,A -85,B 0,C 180,E1 -16393.615,E2 -16393.615} C_VEL
LIN {X 0,Y 298.542,Z 420.795,A -85,B 0,C 180,E1 -16396.408,E2 -16396.408} C_VEL
LIN {X 0,Y 298.505,Z 420.798,A -85,B 0,C 180,E1 -16399.654,E2 -16399.654} C_VEL
LIN {X 0,Y 298.45,Z 420.806,A -85,B 0,C 180,E1 -16403.597,E2 -16403.597} C_VEL
LIN {X 0,Y 298.483,Z 420.803,A -85,B 0,C 180,E1 -16406.574,E2 -16406.574} C_VEL
LIN {X 0,Y 298.414,Z 420.811,A -85,B 0,C 180,E1 -16409.641,E2 -16409.641} C_VEL
LIN {X 0,Y 298.388,Z 420.818,A -85,B 0,C 180,E1 -16412.8,E2 -16412.8} C_VEL
LIN {X 0,Y 298.459,Z 420.809,A -85,B 0,C 180,E1 -16416.812,E2 -16416.812} C_VEL
LIN {X 0,Y 298.445,Z 420.809,A -85,B 0,C 180,E1 -16421.25,E2 -16421.25} C_VEL
LIN {X 0,Y 298.411,Z 420.814,A -85,B 0,C 180,E1 -16425.047,E2 -16425.047} C_VEL
LIN {X 0,Y 298.382,Z 420.818,A -85,B 0,C 180,E1 -16428.912,E2 -16428.912} C_VEL
LIN {X 0,Y 298.459,Z 420.807,A -85,B 0,C 180,E1 -16433.188,E2 -16433.188} C_VEL
LIN {X 0,Y 298.389,Z 420.815,A -85,B 0,C 180,E1 -16437.2,E2 -16437.2} C_VEL
LIN {X 0,Y 298.422,Z 420.814,A -85,B 0,C 180,E1 -16440.617,E2 -16440.617} C_VEL
LIN {X 0,Y 298.473,Z 420.805,A -85,B 0,C 180,E1 -16443.476,E2 -16443.476} C_VEL
LIN {X 0,Y 298.478,Z 420.863,A -85,B 0,C 180,E1 -16445.179,E2 -16445.179} C_VEL
LIN {X 0,Y 299.486,Z 423.7,A -85,B 0,C 180,E1 -16445.342,E2 -16445.342} C_VEL
LIN {X 0,Y 304.007,Z 432.568,A -85,B 0,C 180,E1 -16445.992,E2 -16445.992} C_VEL
LIN {X 0,Y 309.441,Z 440.77,A -85,B 0,C 180,E1 -16446.796,E2 -16446.796} C_VEL
LIN {X 0,Y 313.936,Z 446.705,A -85,B 0,C 180,E1 -16447.517,E2 -16447.517} C_VEL
LIN {X 0,Y 320.29,Z 454.715,A -85,B 0,C 180,E1 -16448.66,E2 -16448.66} C_VEL
LIN {X 0,Y 327.134,Z 462.604,A -85,B 0,C 180,E1 -16450.033,E2 -16450.033} C_VEL
LIN {X 0,Y 332.072,Z 467.975,A -85,B 0,C 180,E1 -16451.115,E2 -16451.115} C_VEL
LIN {X 0,Y 338.632,Z 474.75,A -85,B 0,C 180,E1 -16452.683,E2 -16452.683} C_VEL
LIN {X 0,Y 345.04,Z 480.933,A -85,B 0,C 180,E1 -16454.401,E2 -16454.401} C_VEL
LIN {X 0,Y 348.494,Z 484.451,A -85,B 0,C 180,E1 -16455.464,E2 -16455.464} C_VEL
LIN {X 0,Y 353.369,Z 488.729,A -85,B 0,C 180,E1 -16457.039,E2 -16457.039} C_VEL
LIN {X 0,Y 357.756,Z 492.721,A -85,B 0,C 180,E1 -16458.671,E2 -16458.671} C_VEL
LIN {X 0,Y 360.984,Z 494.922,A -85,B 0,C 180,E1 -16459.909,E2 -16459.909} C_VEL
LIN {X 0,Y 364.275,Z 498.247,A -85,B 0,C 180,E1 -16461.68,E2 -16461.68} C_VEL
LIN {X 0,Y 366.97,Z 500.645,A -85,B 0,C 180,E1 -16463.402,E2 -16463.402} C_VEL
LIN {X 0,Y 368.542,Z 501.669,A -85,B 0,C 180,E1 -16464.529,E2 -16464.529} C_VEL
LIN {X 0,Y 369.925,Z 502.36,A -85,B 0,C 180,E1 -16465.642,E2 -16465.642} C_VEL
LIN {X 0,Y 371.127,Z 502.725,A -85,B 0,C 180,E1 -16466.743,E2 -16466.743} C_VEL
LIN {X 0,Y 372.024,Z 502.932,A -85,B 0,C 180,E1 -16467.835,E2 -16467.835} C_VEL
LIN {X 0,Y 372.573,Z 503.048,A -85,B 0,C 180,E1 -16468.919,E2 -16468.919} C_VEL
LIN {X 0,Y 372.753,Z 503.092,A -85,B 0,C 180,E1 -16470,E2 -16470} C_VEL
LIN {X 0,Y 372.549,Z 503.056,A -85,B 0,C 180,E1 -16471.108,E2 -16471.108} C_VEL
LIN {X 0,Y 371.987,Z 502.969,A -85,B 0,C 180,E1 -16472.165,E2 -16472.165} C_VEL
LIN {X 0,Y 371.125,Z 502.716,A -85,B 0,C 180,E1 -16473.257,E2 -16473.257} C_VEL
LIN {X 0,Y 369.925,Z 502.363,A -85,B 0,C 180,E1 -16474.358,E2 -16474.358} C_VEL
LIN {X 0,Y 367.582,Z 501.066,A -85,B 0,C 180,E1 -16476.172,E2 -16476.172} C_VEL
LIN {X 0,Y 365.201,Z 499.164,A -85,B 0,C 180,E1 -16477.742,E2 -16477.742} C_VEL
LIN {X 0,Y 362.964,Z 496.845,A -85,B 0,C 180,E1 -16479.073,E2 -16479.073} C_VEL
LIN {X 0,Y 360.972,Z 494.913,A -85,B 0,C 180,E1 -16480.092,E2 -16480.092} C_VEL
LIN {X 0,Y 356.276,Z 491.492,A -85,B 0,C 180,E1 -16481.884,E2 -16481.884} C_VEL
LIN {X 0,Y 351.893,Z 487.289,A -85,B 0,C 180,E1 -16483.483,E2 -16483.483} C_VEL
LIN {X 0,Y 347.241,Z 483.206,A -85,B 0,C 180,E1 -16484.932,E2 -16484.932} C_VEL
LIN {X 0,Y 342.191,Z 478.251,A -85,B 0,C 180,E1 -16486.395,E2 -16486.395} C_VEL
LIN {X 0,Y 336.221,Z 472.195,A -85,B 0,C 180,E1 -16487.917,E2 -16487.917} C_VEL
LIN {X 0,Y 330.556,Z 466.216,A -85,B 0,C 180,E1 -16489.244,E2 -16489.244} C_VEL
LIN {X 0,Y 324.712,Z 459.751,A -85,B 0,C 180,E1 -16490.479,E2 -16490.479} C_VEL
LIN {X 0,Y 317.879,Z 451.728,A -85,B 0,C 180,E1 -16491.788,E2 -16491.788} C_VEL
LIN {X 0,Y 311.011,Z 443.029,A -85,B 0,C 180,E1 -16492.953,E2 -16492.953} C_VEL
LIN {X 0,Y 305.23,Z 434.589,A -85,B 0,C 180,E1 -16493.825,E2 -16493.825} C_VEL
LIN {X 0,Y 300.951,Z 426.697,A -85,B 0,C 180,E1 -16494.451,E2 -16494.451} C_VEL
LIN {X 0,Y 298.566,Z 421.392,A -85,B 0,C 180,E1 -16494.799,E2 -16494.799} C_VEL
LIN {X 0,Y 298.464,Z 420.807,A -85,B 0,C 180,E1 -16494.844,E2 -16494.844} C_VEL
LIN {X 0,Y 298.454,Z 420.808,A -85,B 0,C 180,E1 -16498.096,E2 -16498.096} C_VEL
LIN {X 0,Y 298.388,Z 420.816,A -85,B 0,C 180,E1 -16502.016,E2 -16502.016} C_VEL
LIN {X 0,Y 298.426,Z 420.81,A -85,B 0,C 180,E1 -16506.068,E2 -16506.068} C_VEL
LIN {X 0,Y 298.403,Z 420.816,A -85,B 0,C 180,E1 -16509.486,E2 -16509.486} C_VEL
LIN {X 0,Y 298.392,Z 420.817,A -85,B 0,C 180,E1 -16513.103,E2 -16513.103} C_VEL
LIN {X 0,Y 298.396,Z 420.816,A -85,B 0,C 180,E1 -16516.921,E2 -16516.921} C_VEL
LIN {X 0,Y 298.392,Z 420.817,A -85,B 0,C 180,E1 -16521.008,E2 -16521.008} C_VEL
LIN {X 0,Y 298.411,Z 420.811,A -85,B 0,C 180,E1 -16523.93,E2 -16523.93} C_VEL
LIN {X 0,Y 298.388,Z 420.814,A -85,B 0,C 180,E1 -16527.984,E2 -16527.984} C_VEL
LIN {X 0,Y 298.457,Z 420.805,A -85,B 0,C 180,E1 -16531.905,E2 -16531.905} C_VEL
LIN {X 0,Y 298.478,Z 420.805,A -85,B 0,C 180,E1 -16534.924,E2 -16534.924} C_VEL
LIN {X 0,Y 298.443,Z 420.806,A -85,B 0,C 180,E1 -16539.316,E2 -16539.316} C_VEL
LIN {X 0,Y 298.531,Z 420.797,A -85,B 0,C 180,E1 -16542.18,E2 -16542.18} C_VEL
LIN {X 0,Y 298.586,Z 420.79,A -85,B 0,C 180,E1 -16544.995,E2 -16544.995} C_VEL
LIN {X 0,Y 298.584,Z 420.79,A -85,B 0,C 180,E1 -16549.147,E2 -16549.147} C_VEL
LIN {X 0,Y 298.734,Z 420.77,A -85,B 0,C 180,E1 -16551.886,E2 -16551.886} C_VEL
LIN {X 0,Y 298.651,Z 420.784,A -85,B 0,C 180,E1 -16554.6,E2 -16554.6} C_VEL
LIN {X 0,Y 298.917,Z 420.741,A -85,B 0,C 180,E1 -16558.654,E2 -16558.654} C_VEL
LIN {X 0,Y 298.917,Z 420.747,A -85,B 0,C 180,E1 -16561.348,E2 -16561.348} C_VEL
LIN {X 0,Y 298.781,Z 420.768,A -85,B 0,C 180,E1 -16566.755,E2 -16566.755} C_VEL
LIN {X 0,Y 298.731,Z 420.773,A -85,B 0,C 180,E1 -16567.905,E2 -16567.905} C_VEL
LIN {X 0,Y 298.049,Z 420.861,A -85,B 0,C 180,E1 -16569.029,E2 -16569.029} C_VEL
LIN {X 0,Y 295.095,Z 421.227,A -85,B 0,C 180,E1 -16570.856,E2 -16570.856} C_VEL
LIN {X 0,Y 292.608,Z 421.54,A -85,B 0,C 180,E1 -16572.338,E2 -16572.338} C_VEL
LIN {X 0,Y 291.576,Z 421.664,A -85,B 0,C 180,E1 -16573.49,E2 -16573.49} C_VEL
LIN {X 0,Y 291.512,Z 421.673,A -85,B 0,C 180,E1 -16573.88,E2 -16573.88} C_VEL
LIN {X 0,Y 291.481,Z 421.676,A -85,B 0,C 180,E1 -16576.819,E2 -16576.819} C_VEL
LIN {X 0,Y 291.447,Z 421.682,A -85,B 0,C 180,E1 -16579.876,E2 -16579.876} C_VEL
LIN {X 0,Y 291.379,Z 421.693,A -85,B 0,C 180,E1 -16584.208,E2 -16584.208} C_VEL
LIN {X 0,Y 291.419,Z 421.684,A -85,B 0,C 180,E1 -16587.273,E2 -16587.273} C_VEL
LIN {X 0,Y 291.336,Z 421.697,A -85,B 0,C 180,E1 -16590.438,E2 -16590.438} C_VEL
LIN {X 0,Y 291.345,Z 421.699,A -85,B 0,C 180,E1 -16592.406,E2 -16592.406} C_VEL
LIN {X 0,Y 291.547,Z 423.122,A -85,B 0,C 180,E1 -16595.349,E2 -16595.349} C_VEL
LIN {X 0,Y 291.935,Z 425.799,A -85,B 0,C 180,E1 -16599.615,E2 -16599.615} C_VEL
LIN {X 0,Y 292.198,Z 427.657,A -85,B 0,C 180,E1 -16602.336,E2 -16602.336} C_VEL
LIN {X 0,Y 292.436,Z 430.256,A -85,B 0,C 180,E1 -16605.819,E2 -16605.819} C_VEL
LIN {X 0,Y 292.364,Z 432.129,A -85,B 0,C 180,E1 -16608.177,E2 -16608.177} C_VEL
LIN {X 0,Y 292.035,Z 434.761,A -85,B 0,C 180,E1 -16611.267,E2 -16611.267} C_VEL
LIN {X 0,Y 291.484,Z 438.194,A -85,B 0,C 180,E1 -16615.064,E2 -16615.064} C_VEL
LIN {X 0,Y 291.1,Z 440.896,A -85,B 0,C 180,E1 -16617.918,E2 -16617.918} C_VEL
LIN {X 0,Y 290.608,Z 443.948,A -85,B 0,C 180,E1 -16621.075,E2 -16621.075} C_VEL
LIN {X 0,Y 290.186,Z 447.782,A -85,B 0,C 180,E1 -16624.797,E2 -16624.797} C_VEL
LIN {X 0,Y 292.284,Z 455.834,A -85,B 0,C 180,E1 -16625.346,E2 -16625.346} C_VEL
LIN {X 0,Y 294.722,Z 466.032,A -85,B 0,C 180,E1 -16626.178,E2 -16626.178} C_VEL
LIN {X 0,Y 296.38,Z 475.498,A -85,B 0,C 180,E1 -16627.062,E2 -16627.062} C_VEL
LIN {X 0,Y 297.557,Z 484.864,A -85,B 0,C 180,E1 -16628.07,E2 -16628.07} C_VEL
LIN {X 0,Y 298.253,Z 493.413,A -85,B 0,C 180,E1 -16629.126,E2 -16629.126} C_VEL
LIN {X 0,Y 296.963,Z 502.324,A -85,B 0,C 180,E1 -16630.291,E2 -16630.291} C_VEL
LIN {X 0,Y 295.557,Z 510.853,A -85,B 0,C 180,E1 -16631.635,E2 -16631.635} C_VEL
LIN {X 0,Y 294.487,Z 517.427,A -85,B 0,C 180,E1 -16632.86,E2 -16632.86} C_VEL
LIN {X 0,Y 293.265,Z 524.275,A -85,B 0,C 180,E1 -16634.36,E2 -16634.36} C_VEL
LIN {X 0,Y 292.103,Z 530.812,A -85,B 0,C 180,E1 -16636.078,E2 -16636.078} C_VEL
LIN {X 0,Y 291.281,Z 535.313,A -85,B 0,C 180,E1 -16637.459,E2 -16637.459} C_VEL
LIN {X 0,Y 290.461,Z 540.808,A -85,B 0,C 180,E1 -16639.545,E2 -16639.545} C_VEL
LIN {X 0,Y 289.884,Z 545.136,A -85,B 0,C 180,E1 -16641.636,E2 -16641.636} C_VEL
LIN {X 0,Y 289.61,Z 547.503,A -85,B 0,C 180,E1 -16643.031,E2 -16643.031} C_VEL
LIN {X 0,Y 289.432,Z 549.538,A -85,B 0,C 180,E1 -16644.608,E2 -16644.608} C_VEL
LIN {X 0,Y 289.439,Z 551.757,A -85,B 0,C 180,E1 -16647.217,E2 -16647.217} C_VEL
LIN {X 0,Y 289.409,Z 552.346,A -85,B 0,C 180,E1 -16648.609,E2 -16648.609} C_VEL
LIN {X 0,Y 289.409,Z 552.346,A -85,B 0,C 180,E1 -16651.391,E2 -16651.391} C_VEL
LIN {X 0,Y 289.44,Z 551.757,A -85,B 0,C 180,E1 -16652.783,E2 -16652.783} C_VEL
LIN {X 0,Y 289.479,Z 549.305,A -85,B 0,C 180,E1 -16655.573,E2 -16655.573} C_VEL
LIN {X 0,Y 289.731,Z 546.353,A -85,B 0,C 180,E1 -16657.667,E2 -16657.667} C_VEL
LIN {X 0,Y 290.258,Z 542.363,A -85,B 0,C 180,E1 -16659.758,E2 -16659.758} C_VEL
LIN {X 0,Y 290.982,Z 537.23,A -85,B 0,C 180,E1 -16661.847,E2 -16661.847} C_VEL
LIN {X 0,Y 291.896,Z 531.968,A -85,B 0,C 180,E1 -16663.577,E2 -16663.577} C_VEL
LIN {X 0,Y 293.048,Z 525.652,A -85,B 0,C 180,E1 -16665.296,E2 -16665.296} C_VEL
LIN {X 0,Y 294.298,Z 518.601,A -85,B 0,C 180,E1 -16666.894,E2 -16666.894} C_VEL
LIN {X 0,Y 295.486,Z 510.851,A -85,B 0,C 180,E1 -16668.369,E2 -16668.369} C_VEL
LIN {X 0,Y 296.95,Z 502.324,A -85,B 0,C 180,E1 -16669.709,E2 -16669.709} C_VEL
LIN {X 0,Y 298.232,Z 493.412,A -85,B 0,C 180,E1 -16670.876,E2 -16670.876} C_VEL
LIN {X 0,Y 297.112,Z 480.731,A -85,B 0,C 180,E1 -16672.405,E2 -16672.405} C_VEL
LIN {X 0,Y 295.499,Z 469.798,A -85,B 0,C 180,E1 -16673.486,E2 -16673.486} C_VEL
LIN {X 0,Y 292.989,Z 458.452,A -85,B 0,C 180,E1 -16674.451,E2 -16674.451} C_VEL
LIN {X 0,Y 290.281,Z 448.696,A -85,B 0,C 180,E1 -16675.162,E2 -16675.162} C_VEL
LIN {X 0,Y 290.179,Z 447.651,A -85,B 0,C 180,E1 -16675.233,E2 -16675.233} C_VEL
LIN {X 0,Y 290.706,Z 443.352,A -85,B 0,C 180,E1 -16679.502,E2 -16679.502} C_VEL
LIN {X 0,Y 291.124,Z 440.608,A -85,B 0,C 180,E1 -16682.334,E2 -16682.334} C_VEL
LIN {X 0,Y 291.529,Z 437.773,A -85,B 0,C 180,E1 -16685.35,E2 -16685.35} C_VEL
LIN {X 0,Y 292.036,Z 434.751,A -85,B 0,C 180,E1 -16688.733,E2 -16688.733} C_VEL
LIN {X 0,Y 292.385,Z 431.728,A -85,B 0,C 180,E1 -16692.3,E2 -16692.3} C_VEL
LIN {X 0,Y 292.345,Z 429.003,A -85,B 0,C 180,E1 -16695.799,E2 -16695.799} C_VEL
LIN {X 0,Y 292.029,Z 426.397,A -85,B 0,C 180,E1 -16699.474,E2 -16699.474} C_VEL
LIN {X 0,Y 291.684,Z 424.136,A -85,B 0,C 180,E1 -16702.96,E2 -16702.96} C_VEL
LIN {X 0,Y 291.416,Z 422.163,A -85,B 0,C 180,E1 -16706.31,E2 -16706.31} C_VEL
LIN {X 0,Y 291.373,Z 421.696,A -85,B 0,C 180,E1 -16707.95,E2 -16707.95} C_VEL
LIN {X 0,Y 291.379,Z 421.69,A -85,B 0,C 180,E1 -16711.157,E2 -16711.157} C_VEL
LIN {X 0,Y 291.412,Z 421.686,A -85,B 0,C 180,E1 -16714.271,E2 -16714.271} C_VEL
LIN {X 0,Y 291.37,Z 421.691,A -85,B 0,C 180,E1 -16717.298,E2 -16717.298} C_VEL
LIN {X 0,Y 291.454,Z 421.68,A -85,B 0,C 180,E1 -16720.269,E2 -16720.269} C_VEL
LIN {X 0,Y 291.536,Z 421.668,A -85,B 0,C 180,E1 -16724.633,E2 -16724.633} C_VEL
LIN {X 0,Y 291.53,Z 421.669,A -85,B 0,C 180,E1 -16728.88,E2 -16728.88} C_VEL
LIN {X 0,Y 291.682,Z 421.653,A -85,B 0,C 180,E1 -16731.687,E2 -16731.687} C_VEL
LIN {X 0,Y 291.622,Z 421.657,A -85,B 0,C 180,E1 -16734.467,E2 -16734.467} C_VEL
LIN {X 0,Y 291.883,Z 421.623,A -85,B 0,C 180,E1 -16738.62,E2 -16738.62} C_VEL
LIN {X 0,Y 291.883,Z 421.616,A -85,B 0,C 180,E1 -16741.379,E2 -16741.379} C_VEL
LIN {X 0,Y 291.729,Z 421.645,A -85,B 0,C 180,E1 -16746.918,E2 -16746.918} C_VEL
LIN {X 0,Y 291.568,Z 421.664,A -85,B 0,C 180,E1 -16749.713,E2 -16749.713} C_VEL
LIN {X 0,Y 291.515,Z 421.669,A -85,B 0,C 180,E1 -16753.95,E2 -16753.95} C_VEL
LIN {X 0,Y 291.48,Z 421.676,A -85,B 0,C 180,E1 -16756.817,E2 -16756.817} C_VEL
LIN {X 0,Y 291.444,Z 421.677,A -85,B 0,C 180,E1 -16759.874,E2 -16759.874} C_VEL
LIN {X 0,Y 291.393,Z 421.684,A -85,B 0,C 180,E1 -16764.205,E2 -16764.205} C_VEL
LIN {X 0,Y 291.416,Z 421.685,A -85,B 0,C 180,E1 -16767.271,E2 -16767.271} C_VEL
LIN {X 0,Y 291.331,Z 421.695,A -85,B 0,C 180,E1 -16770.437,E2 -16770.437} C_VEL
LIN {X 0,Y 291.338,Z 421.692,A -85,B 0,C 180,E1 -16773.698,E2 -16773.698} C_VEL
LIN {X 0,Y 291.392,Z 421.687,A -85,B 0,C 180,E1 -16777.26,E2 -16777.26} C_VEL
LIN {X 0,Y 291.394,Z 421.689,A -85,B 0,C 180,E1 -16780.631,E2 -16780.631} C_VEL
LIN {X 0,Y 291.347,Z 421.694,A -85,B 0,C 180,E1 -16784.39,E2 -16784.39} C_VEL
LIN {X 0,Y 291.326,Z 421.697,A -85,B 0,C 180,E1 -16788.403,E2 -16788.403} C_VEL
LIN {X 0,Y 291.359,Z 421.692,A -85,B 0,C 180,E1 -16791.16,E2 -16791.16} C_VEL
LIN {X 0,Y 291.38,Z 421.692,A -85,B 0,C 180,E1 -16794.63,E2 -16794.63} C_VEL
LIN {X 0,Y 291.365,Z 421.691,A -85,B 0,C 180,E1 -16797.951,E2 -16797.951} C_VEL
LIN {X 0,Y 291.372,Z 421.69,A -85,B 0,C 180,E1 -16801.158,E2 -16801.158} C_VEL
LIN {X 0,Y 291.439,Z 421.684,A -85,B 0,C 180,E1 -16804.532,E2 -16804.532} C_VEL
LIN {X 0,Y 292.472,Z 424.592,A -85,B 0,C 180,E1 -16804.728,E2 -16804.728} C_VEL
LIN {X 0,Y 297.366,Z 434.634,A -85,B 0,C 180,E1 -16805.496,E2 -16805.496} C_VEL
LIN {X 0,Y 302.219,Z 442.718,A -85,B 0,C 180,E1 -16806.296,E2 -16806.296} C_VEL
LIN {X 0,Y 308.194,Z 450.88,A -85,B 0,C 180,E1 -16807.279,E2 -16807.279} C_VEL
LIN {X 0,Y 315.246,Z 459.655,A -85,B 0,C 180,E1 -16808.541,E2 -16808.541} C_VEL
LIN {X 0,Y 321.852,Z 467.292,A -85,B 0,C 180,E1 -16809.874,E2 -16809.874} C_VEL
LIN {X 0,Y 328.138,Z 474.111,A -85,B 0,C 180,E1 -16811.261,E2 -16811.261} C_VEL
LIN {X 0,Y 333.509,Z 479.599,A -85,B 0,C 180,E1 -16812.548,E2 -16812.548} C_VEL
LIN {X 0,Y 338.94,Z 484.824,A -85,B 0,C 180,E1 -16813.977,E2 -16813.977} C_VEL
LIN {X 0,Y 343.408,Z 489.392,A -85,B 0,C 180,E1 -16815.335,E2 -16815.335} C_VEL
LIN {X 0,Y 348.135,Z 493.5,A -85,B 0,C 180,E1 -16816.841,E2 -16816.841} C_VEL
LIN {X 0,Y 352.637,Z 497.664,A -85,B 0,C 180,E1 -16818.504,E2 -16818.504} C_VEL
LIN {X 0,Y 356.695,Z 500.624,A -85,B 0,C 180,E1 -16820.11,E2 -16820.11} C_VEL
LIN {X 0,Y 359.355,Z 503.316,A -85,B 0,C 180,E1 -16821.566,E2 -16821.566} C_VEL
LIN {X 0,Y 362.092,Z 505.802,A -85,B 0,C 180,E1 -16823.313,E2 -16823.313} C_VEL
LIN {X 0,Y 363.711,Z 506.893,A -85,B 0,C 180,E1 -16824.456,E2 -16824.456} C_VEL
LIN {X 0,Y 366.147,Z 508.011,A -85,B 0,C 180,E1 -16826.466,E2 -16826.466} C_VEL
LIN {X 0,Y 367.359,Z 508.32,A -85,B 0,C 180,E1 -16827.807,E2 -16827.807} C_VEL
LIN {X 0,Y 367.968,Z 508.434,A -85,B 0,C 180,E1 -16828.906,E2 -16828.906} C_VEL
LIN {X 0,Y 368.147,Z 508.496,A -85,B 0,C 180,E1 -16830,E2 -16830} C_VEL
LIN {X 0,Y 367.939,Z 508.461,A -85,B 0,C 180,E1 -16831.094,E2 -16831.094} C_VEL
LIN {X 0,Y 367.335,Z 508.338,A -85,B 0,C 180,E1 -16832.193,E2 -16832.193} C_VEL
LIN {X 0,Y 366.147,Z 508.007,A -85,B 0,C 180,E1 -16833.534,E2 -16833.534} C_VEL
LIN {X 0,Y 363.735,Z 506.895,A -85,B 0,C 180,E1 -16835.544,E2 -16835.544} C_VEL
LIN {X 0,Y 361.29,Z 505.135,A -85,B 0,C 180,E1 -16837.223,E2 -16837.223} C_VEL
LIN {X 0,Y 358.342,Z 502.268,A -85,B 0,C 180,E1 -16839.027,E2 -16839.027} C_VEL
LIN {X 0,Y 355.923,Z 500,A -85,B 0,C 180,E1 -16840.236,E2 -16840.236} C_VEL
LIN {X 0,Y 351.81,Z 497.013,A -85,B 0,C 180,E1 -16841.807,E2 -16841.807} C_VEL
LIN {X 0,Y 347.004,Z 492.44,A -85,B 0,C 180,E1 -16843.555,E2 -16843.555} C_VEL
LIN {X 0,Y 342.095,Z 488.083,A -85,B 0,C 180,E1 -16845.082,E2 -16845.082} C_VEL
LIN {X 0,Y 337.163,Z 483.243,A -85,B 0,C 180,E1 -16846.497,E2 -16846.497} C_VEL
LIN {X 0,Y 330.799,Z 476.812,A -85,B 0,C 180,E1 -16848.12,E2 -16848.12} C_VEL
LIN {X 0,Y 324.823,Z 470.424,A -85,B 0,C 180,E1 -16849.506,E2 -16849.506} C_VEL
LIN {X 0,Y 318.137,Z 462.944,A -85,B 0,C 180,E1 -16850.907,E2 -16850.907} C_VEL
LIN {X 0,Y 311.199,Z 454.719,A -85,B 0,C 180,E1 -16852.194,E2 -16852.194} C_VEL
LIN {X 0,Y 304.837,Z 446.333,A -85,B 0,C 180,E1 -16853.28,E2 -16853.28} C_VEL
LIN {X 0,Y 298.84,Z 437.369,A -85,B 0,C 180,E1 -16854.259,E2 -16854.259} C_VEL
LIN {X 0,Y 294.432,Z 428.813,A -85,B 0,C 180,E1 -16854.97,E2 -16854.97} C_VEL
LIN {X 0,Y 291.617,Z 422.631,A -85,B 0,C 180,E1 -16855.404,E2 -16855.404} C_VEL
LIN {X 0,Y 291.428,Z 421.686,A -85,B 0,C 180,E1 -16855.498,E2 -16855.498} C_VEL
LIN {X 0,Y 291.372,Z 421.69,A -85,B 0,C 180,E1 -16858.842,E2 -16858.842} C_VEL
LIN {X 0,Y 291.337,Z 421.693,A -85,B 0,C 180,E1 -16862.403,E2 -16862.403} C_VEL
LIN {X 0,Y 291.38,Z 421.692,A -85,B 0,C 180,E1 -16865.37,E2 -16865.37} C_VEL
LIN {X 0,Y 291.359,Z 421.692,A -85,B 0,C 180,E1 -16868.84,E2 -16868.84} C_VEL
LIN {X 0,Y 291.313,Z 421.696,A -85,B 0,C 180,E1 -16872.492,E2 -16872.492} C_VEL
LIN {X 0,Y 291.313,Z 421.696,A -85,B 0,C 180,E1 -16876.364,E2 -16876.364} C_VEL
LIN {X 0,Y 291.372,Z 421.689,A -85,B 0,C 180,E1 -16880.519,E2 -16880.519} C_VEL
LIN {X 0,Y 291.397,Z 421.688,A -85,B 0,C 180,E1 -16882.919,E2 -16882.919} C_VEL
LIN {X 0,Y 291.338,Z 421.692,A -85,B 0,C 180,E1 -16886.302,E2 -16886.302} C_VEL
LIN {X 0,Y 291.38,Z 421.687,A -85,B 0,C 180,E1 -16890.26,E2 -16890.26} C_VEL
LIN {X 0,Y 291.41,Z 421.683,A -85,B 0,C 180,E1 -16894.272,E2 -16894.272} C_VEL
LIN {X 0,Y 291.374,Z 421.69,A -85,B 0,C 180,E1 -16897.3,E2 -16897.3} C_VEL
LIN {X 0,Y 291.451,Z 421.676,A -85,B 0,C 180,E1 -16900.271,E2 -16900.271} C_VEL
LIN {X 0,Y 291.534,Z 421.67,A -85,B 0,C 180,E1 -16904.635,E2 -16904.635} C_VEL
LIN {X 0,Y 291.528,Z 421.671,A -85,B 0,C 180,E1 -16908.881,E2 -16908.881} C_VEL
LIN {X 0,Y 291.681,Z 421.649,A -85,B 0,C 180,E1 -16911.688,E2 -16911.688} C_VEL
LIN {X 0,Y 291.621,Z 421.661,A -85,B 0,C 180,E1 -16914.469,E2 -16914.469} C_VEL
LIN {X 0,Y 291.883,Z 421.616,A -85,B 0,C 180,E1 -16918.621,E2 -16918.621} C_VEL
LIN {X 0,Y 291.883,Z 421.623,A -85,B 0,C 180,E1 -16921.38,E2 -16921.38} C_VEL
LIN {X 0,Y 291.73,Z 421.645,A -85,B 0,C 180,E1 -16926.919,E2 -16926.919} C_VEL
LIN {X 0,Y 291.569,Z 421.665,A -85,B 0,C 180,E1 -16929.715,E2 -16929.715} C_VEL
LIN {X 0,Y 291.512,Z 421.673,A -85,B 0,C 180,E1 -16933.88,E2 -16933.88} C_VEL
LIN {X 0,Y 290.877,Z 421.756,A -85,B 0,C 180,E1 -16935.032,E2 -16935.032} C_VEL
LIN {X 0,Y 287.967,Z 422.115,A -85,B 0,C 180,E1 -16936.906,E2 -16936.906} C_VEL
LIN {X 0,Y 285.487,Z 422.425,A -85,B 0,C 180,E1 -16938.429,E2 -16938.429} C_VEL
LIN {X 0,Y 284.448,Z 422.552,A -85,B 0,C 180,E1 -16939.61,E2 -16939.61} C_VEL
LIN {X 0,Y 284.379,Z 422.562,A -85,B 0,C 180,E1 -16940.011,E2 -16940.011} C_VEL
LIN {X 0,Y 284.331,Z 422.57,A -85,B 0,C 180,E1 -16943.861,E2 -16943.861} C_VEL
LIN {X 0,Y 284.394,Z 422.559,A -85,B 0,C 180,E1 -16947.175,E2 -16947.175} C_VEL
LIN {X 0,Y 284.296,Z 422.575,A -85,B 0,C 180,E1 -16951.275,E2 -16951.275} C_VEL
LIN {X 0,Y 284.336,Z 422.872,A -85,B 0,C 180,E1 -16952.942,E2 -16952.942} C_VEL
LIN {X 0,Y 284.588,Z 424.805,A -85,B 0,C 180,E1 -16956.349,E2 -16956.349} C_VEL
LIN {X 0,Y 284.963,Z 427.165,A -85,B 0,C 180,E1 -16960.135,E2 -16960.135} C_VEL
LIN {X 0,Y 285.286,Z 429.546,A -85,B 0,C 180,E1 -16963.613,E2 -16963.613} C_VEL
LIN {X 0,Y 285.371,Z 431.624,A -85,B 0,C 180,E1 -16966.405,E2 -16966.405} C_VEL
LIN {X 0,Y 285.171,Z 434.357,A -85,B 0,C 180,E1 -16969.818,E2 -16969.818} C_VEL
LIN {X 0,Y 284.611,Z 437.677,A -85,B 0,C 180,E1 -16973.656,E2 -16973.656} C_VEL
LIN {X 0,Y 284.117,Z 440.931,A -85,B 0,C 180,E1 -16977.251,E2 -16977.251} C_VEL
LIN {X 0,Y 283.636,Z 443.795,A -85,B 0,C 180,E1 -16980.294,E2 -16980.294} C_VEL
LIN {X 0,Y 283.162,Z 447.479,A -85,B 0,C 180,E1 -16984.102,E2 -16984.102} C_VEL
LIN {X 0,Y 286.869,Z 461.839,A -85,B 0,C 180,E1 -16985.194,E2 -16985.194} C_VEL
LIN {X 0,Y 289.158,Z 472.778,A -85,B 0,C 180,E1 -16986.22,E2 -16986.22} C_VEL
LIN {X 0,Y 290.568,Z 483.58,A -85,B 0,C 180,E1 -16987.392,E2 -16987.392} C_VEL
LIN {X 0,Y 291.34,Z 493.316,A -85,B 0,C 180,E1 -16988.621,E2 -16988.621} C_VEL
LIN {X 0,Y 291.292,Z 495.887,A -85,B 0,C 180,E1 -16988.969,E2 -16988.969} C_VEL
LIN {X 0,Y 289.865,Z 504.395,A -85,B 0,C 180,E1 -16990.158,E2 -16990.158} C_VEL
LIN {X 0,Y 288.428,Z 512.574,A -85,B 0,C 180,E1 -16991.533,E2 -16991.533} C_VEL
LIN {X 0,Y 287.009,Z 521.13,A -85,B 0,C 180,E1 -16993.279,E2 -16993.279} C_VEL
LIN {X 0,Y 285.438,Z 529.459,A -85,B 0,C 180,E1 -16995.382,E2 -16995.382} C_VEL
LIN {X 0,Y 284.327,Z 535.115,A -85,B 0,C 180,E1 -16997.147,E2 -16997.147} C_VEL
LIN {X 0,Y 283.446,Z 540.61,A -85,B 0,C 180,E1 -16999.283,E2 -16999.283} C_VEL
LIN {X 0,Y 282.829,Z 544.938,A -85,B 0,C 180,E1 -17001.426,E2 -17001.426} C_VEL
LIN {X 0,Y 282.558,Z 547.306,A -85,B 0,C 180,E1 -17002.856,E2 -17002.856} C_VEL
LIN {X 0,Y 282.341,Z 549.589,A -85,B 0,C 180,E1 -17004.676,E2 -17004.676} C_VEL
LIN {X 0,Y 282.347,Z 551.56,A -85,B 0,C 180,E1 -17007.147,E2 -17007.147} C_VEL
LIN {X 0,Y 282.333,Z 552.149,A -85,B 0,C 180,E1 -17008.574,E2 -17008.574} C_VEL
LIN {X 0,Y 282.333,Z 552.149,A -85,B 0,C 180,E1 -17011.426,E2 -17011.426} C_VEL
LIN {X 0,Y 282.347,Z 551.56,A -85,B 0,C 180,E1 -17012.853,E2 -17012.853} C_VEL
LIN {X 0,Y 282.388,Z 549.107,A -85,B 0,C 180,E1 -17015.713,E2 -17015.713} C_VEL
LIN {X 0,Y 282.687,Z 546.156,A -85,B 0,C 180,E1 -17017.859,E2 -17017.859} C_VEL
LIN {X 0,Y 283.222,Z 542.165,A -85,B 0,C 180,E1 -17020.003,E2 -17020.003} C_VEL
LIN {X 0,Y 283.984,Z 537.032,A -85,B 0,C 180,E1 -17022.143,E2 -17022.143} C_VEL
LIN {X 0,Y 284.979,Z 531.771,A -85,B 0,C 180,E1 -17023.913,E2 -17023.913} C_VEL
LIN {X 0,Y 286.155,Z 525.453,A -85,B 0,C 180,E1 -17025.673,E2 -17025.673} C_VEL
LIN {X 0,Y 287.298,Z 519.504,A -85,B 0,C 180,E1 -17027.07,E2 -17027.07} C_VEL
LIN {X 0,Y 288.39,Z 512.573,A -85,B 0,C 180,E1 -17028.47,E2 -17028.47} C_VEL
LIN {X 0,Y 289.85,Z 504.395,A -85,B 0,C 180,E1 -17029.843,E2 -17029.843} C_VEL
LIN {X 0,Y 291.259,Z 495.886,A -85,B 0,C 180,E1 -17031.034,E2 -17031.034} C_VEL
LIN {X 0,Y 291.218,Z 490.863,A -85,B 0,C 180,E1 -17031.72,E2 -17031.72} C_VEL
LIN {X 0,Y 290.167,Z 480.035,A -85,B 0,C 180,E1 -17033.017,E2 -17033.017} C_VEL
LIN {X 0,Y 288.609,Z 469.983,A -85,B 0,C 180,E1 -17034.052,E2 -17034.052} C_VEL
LIN {X 0,Y 286.033,Z 458.365,A -85,B 0,C 180,E1 -17035.079,E2 -17035.079} C_VEL
LIN {X 0,Y 283.29,Z 448.58,A -85,B 0,C 180,E1 -17035.824,E2 -17035.824} C_VEL
LIN {X 0,Y 283.164,Z 447.483,A -85,B 0,C 180,E1 -17035.896,E2 -17035.896} C_VEL
LIN {X 0,Y 283.683,Z 443.582,A -85,B 0,C 180,E1 -17039.876,E2 -17039.876} C_VEL
LIN {X 0,Y 284.13,Z 440.694,A -85,B 0,C 180,E1 -17042.967,E2 -17042.967} C_VEL
LIN {X 0,Y 284.608,Z 437.638,A -85,B 0,C 180,E1 -17046.344,E2 -17046.344} C_VEL
LIN {X 0,Y 285.172,Z 434.356,A -85,B 0,C 180,E1 -17050.182,E2 -17050.182} C_VEL
LIN {X 0,Y 285.382,Z 431.612,A -85,B 0,C 180,E1 -17053.593,E2 -17053.593} C_VEL
LIN {X 0,Y 285.25,Z 429.556,A -85,B 0,C 180,E1 -17056.38,E2 -17056.38} C_VEL
LIN {X 0,Y 284.93,Z 427.004,A -85,B 0,C 180,E1 -17060.11,E2 -17060.11} C_VEL
LIN {X 0,Y 284.585,Z 424.799,A -85,B 0,C 180,E1 -17063.651,E2 -17063.651} C_VEL
LIN {X 0,Y 284.317,Z 422.804,A -85,B 0,C 180,E1 -17067.185,E2 -17067.185} C_VEL
LIN {X 0,Y 284.357,Z 422.566,A -85,B 0,C 180,E1 -17070.375,E2 -17070.375} C_VEL
LIN {X 0,Y 284.374,Z 422.564,A -85,B 0,C 180,E1 -17073.585,E2 -17073.585} C_VEL
LIN {X 0,Y 284.329,Z 422.567,A -85,B 0,C 180,E1 -17076.703,E2 -17076.703} C_VEL
LIN {X 0,Y 284.395,Z 422.559,A -85,B 0,C 180,E1 -17081.26,E2 -17081.26} C_VEL
LIN {X 0,Y 284.474,Z 422.548,A -85,B 0,C 180,E1 -17084.469,E2 -17084.469} C_VEL
LIN {X 0,Y 284.482,Z 422.547,A -85,B 0,C 180,E1 -17088.6,E2 -17088.6} C_VEL
LIN {X 0,Y 284.634,Z 422.531,A -85,B 0,C 180,E1 -17091.48,E2 -17091.48} C_VEL
LIN {X 0,Y 284.592,Z 422.533,A -85,B 0,C 180,E1 -17094.33,E2 -17094.33} C_VEL
LIN {X 0,Y 284.849,Z 422.499,A -85,B 0,C 180,E1 -17098.585,E2 -17098.585} C_VEL
LIN {X 0,Y 284.849,Z 422.49,A -85,B 0,C 180,E1 -17101.413,E2 -17101.413} C_VEL
LIN {X 0,Y 284.68,Z 422.524,A -85,B 0,C 180,E1 -17107.09,E2 -17107.09} C_VEL
LIN {X 0,Y 284.512,Z 422.541,A -85,B 0,C 180,E1 -17109.956,E2 -17109.956} C_VEL
LIN {X 0,Y 284.471,Z 422.545,A -85,B 0,C 180,E1 -17114.302,E2 -17114.302} C_VEL
LIN {X 0,Y 284.418,Z 422.559,A -85,B 0,C 180,E1 -17117.248,E2 -17117.248} C_VEL
LIN {X 0,Y 284.372,Z 422.557,A -85,B 0,C 180,E1 -17120.242,E2 -17120.242} C_VEL
LIN {X 0,Y 284.362,Z 422.56,A -85,B 0,C 180,E1 -17123.875,E2 -17123.875} C_VEL
LIN {X 0,Y 284.391,Z 422.561,A -85,B 0,C 180,E1 -17127.173,E2 -17127.173} C_VEL
LIN {X 0,Y 284.289,Z 422.573,A -85,B 0,C 180,E1 -17131.274,E2 -17131.274} C_VEL
LIN {X 0,Y 284.355,Z 422.563,A -85,B 0,C 180,E1 -17135.354,E2 -17135.354} C_VEL
LIN {X 0,Y 284.325,Z 422.566,A -85,B 0,C 180,E1 -17138.166,E2 -17138.166} C_VEL
LIN {X 0,Y 284.334,Z 422.566,A -85,B 0,C 180,E1 -17142.14,E2 -17142.14} C_VEL
LIN {X 0,Y 284.291,Z 422.572,A -85,B 0,C 180,E1 -17146.197,E2 -17146.197} C_VEL
LIN {X 0,Y 284.301,Z 422.57,A -85,B 0,C 180,E1 -17150.024,E2 -17150.024} C_VEL
LIN {X 0,Y 284.345,Z 422.564,A -85,B 0,C 180,E1 -17153.617,E2 -17153.617} C_VEL
LIN {X 0,Y 284.302,Z 422.571,A -85,B 0,C 180,E1 -17157.19,E2 -17157.19} C_VEL
LIN {X 0,Y 284.35,Z 422.567,A -85,B 0,C 180,E1 -17160.376,E2 -17160.376} C_VEL
LIN {X 0,Y 284.381,Z 422.623,A -85,B 0,C 180,E1 -17163.895,E2 -17163.895} C_VEL
LIN {X 0,Y 285.538,Z 425.653,A -85,B 0,C 180,E1 -17164.093,E2 -17164.093} C_VEL
LIN {X 0,Y 291.674,Z 438.424,A -85,B 0,C 180,E1 -17165.141,E2 -17165.141} C_VEL
LIN {X 0,Y 296.645,Z 446.935,A -85,B 0,C 180,E1 -17166.059,E2 -17166.059} C_VEL
LIN {X 0,Y 303.014,Z 455.722,A -85,B 0,C 180,E1 -17167.21,E2 -17167.21} C_VEL
LIN {X 0,Y 311.237,Z 465.9,A -85,B 0,C 180,E1 -17168.749,E2 -17168.749} C_VEL
LIN {X 0,Y 319.238,Z 474.838,A -85,B 0,C 180,E1 -17170.395,E2 -17170.395} C_VEL
LIN {X 0,Y 325.435,Z 481.467,A -85,B 0,C 180,E1 -17171.841,E2 -17171.841} C_VEL
LIN {X 0,Y 331.862,Z 488.004,A -85,B 0,C 180,E1 -17173.476,E2 -17173.476} C_VEL
LIN {X 0,Y 337.409,Z 493.395,A -85,B 0,C 180,E1 -17175.068,E2 -17175.068} C_VEL
LIN {X 0,Y 341.315,Z 496.857,A -85,B 0,C 180,E1 -17176.277,E2 -17176.277} C_VEL
LIN {X 0,Y 346.964,Z 502.107,A -85,B 0,C 180,E1 -17178.314,E2 -17178.314} C_VEL
LIN {X 0,Y 350.322,Z 504.644,A -85,B 0,C 180,E1 -17179.598,E2 -17179.598} C_VEL
LIN {X 0,Y 352.934,Z 506.84,A -85,B 0,C 180,E1 -17180.834,E2 -17180.834} C_VEL
LIN {X 0,Y 354.915,Z 508.938,A -85,B 0,C 180,E1 -17182.033,E2 -17182.033} C_VEL
LIN {X 0,Y 356.771,Z 510.547,A -85,B 0,C 180,E1 -17183.212,E2 -17183.212} C_VEL
LIN {X 0,Y 359.644,Z 512.394,A -85,B 0,C 180,E1 -17185.277,E2 -17185.277} C_VEL
LIN {X 0,Y 361.261,Z 513.04,A -85,B 0,C 180,E1 -17186.654,E2 -17186.654} C_VEL
LIN {X 0,Y 362.28,Z 513.323,A -85,B 0,C 180,E1 -17187.776,E2 -17187.776} C_VEL
LIN {X 0,Y 362.93,Z 513.445,A -85,B 0,C 180,E1 -17188.89,E2 -17188.89} C_VEL
LIN {X 0,Y 363.131,Z 513.497,A -85,B 0,C 180,E1 -17190,E2 -17190} C_VEL
LIN {X 0,Y 362.906,Z 513.465,A -85,B 0,C 180,E1 -17191.11,E2 -17191.11} C_VEL
LIN {X 0,Y 362.254,Z 513.339,A -85,B 0,C 180,E1 -17192.224,E2 -17192.224} C_VEL
LIN {X 0,Y 361.26,Z 513.035,A -85,B 0,C 180,E1 -17193.346,E2 -17193.346} C_VEL
LIN {X 0,Y 359.651,Z 512.385,A -85,B 0,C 180,E1 -17194.735,E2 -17194.735} C_VEL
LIN {X 0,Y 356.764,Z 510.539,A -85,B 0,C 180,E1 -17196.788,E2 -17196.788} C_VEL
LIN {X 0,Y 354.862,Z 508.841,A -85,B 0,C 180,E1 -17198.016,E2 -17198.016} C_VEL
LIN {X 0,Y 352.037,Z 506.01,A -85,B 0,C 180,E1 -17199.606,E2 -17199.606} C_VEL
LIN {X 0,Y 350.188,Z 504.529,A -85,B 0,C 180,E1 -17200.461,E2 -17200.461} C_VEL
LIN {X 0,Y 345.272,Z 500.634,A -85,B 0,C 180,E1 -17202.305,E2 -17202.305} C_VEL
LIN {X 0,Y 342.313,Z 497.735,A -85,B 0,C 180,E1 -17203.403,E2 -17203.403} C_VEL
LIN {X 0,Y 337.579,Z 493.558,A -85,B 0,C 180,E1 -17204.881,E2 -17204.881} C_VEL
LIN {X 0,Y 331.873,Z 487.965,A -85,B 0,C 180,E1 -17206.524,E2 -17206.524} C_VEL
LIN {X 0,Y 325.442,Z 481.477,A -85,B 0,C 180,E1 -17208.163,E2 -17208.163} C_VEL
LIN {X 0,Y 319.218,Z 474.827,A -85,B 0,C 180,E1 -17209.608,E2 -17209.608} C_VEL
LIN {X 0,Y 311.842,Z 466.558,A -85,B 0,C 180,E1 -17211.136,E2 -17211.136} C_VEL
LIN {X 0,Y 303.013,Z 455.726,A -85,B 0,C 180,E1 -17212.789,E2 -17212.789} C_VEL
LIN {X 0,Y 296.128,Z 446.086,A -85,B 0,C 180,E1 -17214.04,E2 -17214.04} C_VEL
LIN {X 0,Y 291,Z 437.282,A -85,B 0,C 180,E1 -17214.971,E2 -17214.971} C_VEL
LIN {X 0,Y 284.544,Z 423.467,A -85,B 0,C 180,E1 -17216.066,E2 -17216.066} C_VEL
LIN {X 0,Y 284.379,Z 422.562,A -85,B 0,C 180,E1 -17216.134,E2 -17216.134} C_VEL
LIN {X 0,Y 284.306,Z 422.57,A -85,B 0,C 180,E1 -17220.097,E2 -17220.097} C_VEL
LIN {X 0,Y 284.3,Z 422.571,A -85,B 0,C 180,E1 -17222.945,E2 -17222.945} C_VEL
LIN {X 0,Y 284.345,Z 422.564,A -85,B 0,C 180,E1 -17226.383,E2 -17226.383} C_VEL
LIN {X 0,Y 284.3,Z 422.57,A -85,B 0,C 180,E1 -17229.994,E2 -17229.994} C_VEL
LIN {X 0,Y 284.259,Z 422.574,A -85,B 0,C 180,E1 -17234.195,E2 -17234.195} C_VEL
LIN {X 0,Y 284.266,Z 422.574,A -85,B 0,C 180,E1 -17238.124,E2 -17238.124} C_VEL
LIN {X 0,Y 284.312,Z 422.567,A -85,B 0,C 180,E1 -17242.279,E2 -17242.279} C_VEL
LIN {X 0,Y 284.302,Z 422.572,A -85,B 0,C 180,E1 -17245.351,E2 -17245.351} C_VEL
LIN {X 0,Y 284.289,Z 422.573,A -85,B 0,C 180,E1 -17248.726,E2 -17248.726} C_VEL
LIN {X 0,Y 284.391,Z 422.561,A -85,B 0,C 180,E1 -17252.827,E2 -17252.827} C_VEL
LIN {X 0,Y 284.359,Z 422.563,A -85,B 0,C 180,E1 -17256.707,E2 -17256.707} C_VEL
LIN {X 0,Y 284.397,Z 422.558,A -85,B 0,C 180,E1 -17261.262,E2 -17261.262} C_VEL
LIN {X 0,Y 284.471,Z 422.55,A -85,B 0,C 180,E1 -17264.47,E2 -17264.47} C_VEL
LIN {X 0,Y 284.48,Z 422.551,A -85,B 0,C 180,E1 -17268.602,E2 -17268.602} C_VEL
LIN {X 0,Y 284.632,Z 422.527,A -85,B 0,C 180,E1 -17271.481,E2 -17271.481} C_VEL
LIN {X 0,Y 284.592,Z 422.535,A -85,B 0,C 180,E1 -17274.332,E2 -17274.332} C_VEL
LIN {X 0,Y 284.849,Z 422.49,A -85,B 0,C 180,E1 -17278.587,E2 -17278.587} C_VEL
LIN {X 0,Y 284.849,Z 422.499,A -85,B 0,C 180,E1 -17281.415,E2 -17281.415} C_VEL
LIN {X 0,Y 284.681,Z 422.522,A -85,B 0,C 180,E1 -17287.091,E2 -17287.091} C_VEL
LIN {X 0,Y 284.514,Z 422.545,A -85,B 0,C 180,E1 -17289.958,E2 -17289.958} C_VEL
LIN {X 0,Y 284.473,Z 422.553,A -85,B 0,C 180,E1 -17294.304,E2 -17294.304} C_VEL
LIN {X 0,Y 284.418,Z 422.555,A -85,B 0,C 180,E1 -17297.25,E2 -17297.25} C_VEL
LIN {X 0,Y 284.379,Z 422.562,A -85,B 0,C 180,E1 -17300.011,E2 -17300.011} C_VEL
LIN {X 0,Y 283.742,Z 422.648,A -85,B 0,C 180,E1 -17301.193,E2 -17301.193} C_VEL
LIN {X 0,Y 280.863,Z 423.007,A -85,B 0,C 180,E1 -17303.118,E2 -17303.118} C_VEL
LIN {X 0,Y 278.409,Z 423.307,A -85,B 0,C 180,E1 -17304.682,E2 -17304.682} C_VEL
LIN {X 0,Y 277.375,Z 423.437,A -85,B 0,C 180,E1 -17305.895,E2 -17305.895} C_VEL
LIN {X 0,Y 277.303,Z 423.44,A -85,B 0,C 180,E1 -17306.306,E2 -17306.306} C_VEL
LIN {X 0,Y 277.27,Z 423.45,A -85,B 0,C 180,E1 -17310.483,E2 -17310.483} C_VEL
LIN {X 0,Y 277.257,Z 423.574,A -85,B 0,C 180,E1 -17312.163,E2 -17312.163} C_VEL
LIN {X 0,Y 277.532,Z 425.597,A -85,B 0,C 180,E1 -17315.872,E2 -17315.872} C_VEL
LIN {X 0,Y 277.838,Z 427.62,A -85,B 0,C 180,E1 -17319.227,E2 -17319.227} C_VEL
LIN {X 0,Y 278.199,Z 430.094,A -85,B 0,C 180,E1 -17323.008,E2 -17323.008} C_VEL
LIN {X 0,Y 278.322,Z 431.501,A -85,B 0,C 180,E1 -17325.007,E2 -17325.007} C_VEL
LIN {X 0,Y 278.306,Z 433.055,A -85,B 0,C 180,E1 -17327.083,E2 -17327.083} C_VEL
LIN {X 0,Y 277.957,Z 436.013,A -85,B 0,C 180,E1 -17330.795,E2 -17330.795} C_VEL
LIN {X 0,Y 277.461,Z 439.084,A -85,B 0,C 180,E1 -17334.369,E2 -17334.369} C_VEL
LIN {X 0,Y 276.928,Z 442.091,A -85,B 0,C 180,E1 -17337.796,E2 -17337.796} C_VEL
LIN {X 0,Y 276.394,Z 445.18,A -85,B 0,C 180,E1 -17341.111,E2 -17341.111} C_VEL
LIN {X 0,Y 276.153,Z 447.319,A -85,B 0,C 180,E1 -17343.414,E2 -17343.414} C_VEL
LIN {X 0,Y 278.232,Z 455.146,A -85,B 0,C 180,E1 -17343.996,E2 -17343.996} C_VEL
LIN {X 0,Y 280.804,Z 465.352,A -85,B 0,C 180,E1 -17344.899,E2 -17344.899} C_VEL
LIN {X 0,Y 282.686,Z 475.208,A -85,B 0,C 180,E1 -17345.895,E2 -17345.895} C_VEL
LIN {X 0,Y 283.801,Z 484.438,A -85,B 0,C 180,E1 -17346.946,E2 -17346.946} C_VEL
LIN {X 0,Y 284.503,Z 493.222,A -85,B 0,C 180,E1 -17348.096,E2 -17348.096} C_VEL
LIN {X 0,Y 284.436,Z 497.04,A -85,B 0,C 180,E1 -17348.627,E2 -17348.627} C_VEL
LIN {X 0,Y 282.433,Z 508.538,A -85,B 0,C 180,E1 -17350.371,E2 -17350.371} C_VEL
LIN {X 0,Y 280.83,Z 516.985,A -85,B 0,C 180,E1 -17351.988,E2 -17351.988} C_VEL
LIN {X 0,Y 279.557,Z 523.879,A -85,B 0,C 180,E1 -17353.572,E2 -17353.572} C_VEL
LIN {X 0,Y 278.297,Z 530.417,A -85,B 0,C 180,E1 -17355.373,E2 -17355.373} C_VEL
LIN {X 0,Y 277.378,Z 534.917,A -85,B 0,C 180,E1 -17356.819,E2 -17356.819} C_VEL
LIN {X 0,Y 276.445,Z 540.412,A -85,B 0,C 180,E1 -17359.008,E2 -17359.008} C_VEL
LIN {X 0,Y 275.796,Z 544.74,A -85,B 0,C 180,E1 -17361.205,E2 -17361.205} C_VEL
LIN {X 0,Y 275.498,Z 547.109,A -85,B 0,C 180,E1 -17362.672,E2 -17362.672} C_VEL
LIN {X 0,Y 275.239,Z 549.625,A -85,B 0,C 180,E1 -17364.776,E2 -17364.776} C_VEL
LIN {X 0,Y 275.256,Z 551.362,A -85,B 0,C 180,E1 -17367.073,E2 -17367.073} C_VEL
LIN {X 0,Y 275.258,Z 551.953,A -85,B 0,C 180,E1 -17368.537,E2 -17368.537} C_VEL
LIN {X 0,Y 275.258,Z 551.953,A -85,B 0,C 180,E1 -17371.463,E2 -17371.463} C_VEL
LIN {X 0,Y 275.257,Z 551.362,A -85,B 0,C 180,E1 -17372.927,E2 -17372.927} C_VEL
LIN {X 0,Y 275.302,Z 548.91,A -85,B 0,C 180,E1 -17375.861,E2 -17375.861} C_VEL
LIN {X 0,Y 275.619,Z 545.958,A -85,B 0,C 180,E1 -17378.062,E2 -17378.062} C_VEL
LIN {X 0,Y 276.204,Z 541.967,A -85,B 0,C 180,E1 -17380.26,E2 -17380.26} C_VEL
LIN {X 0,Y 277.008,Z 536.834,A -85,B 0,C 180,E1 -17382.454,E2 -17382.454} C_VEL
LIN {X 0,Y 278.046,Z 531.572,A -85,B 0,C 180,E1 -17384.267,E2 -17384.267} C_VEL
LIN {X 0,Y 279.277,Z 525.255,A -85,B 0,C 180,E1 -17386.07,E2 -17386.07} C_VEL
LIN {X 0,Y 280.601,Z 518.498,A -85,B 0,C 180,E1 -17387.677,E2 -17387.677} C_VEL
LIN {X 0,Y 281.978,Z 510.455,A -85,B 0,C 180,E1 -17389.283,E2 -17389.283} C_VEL
LIN {X 0,Y 283.565,Z 501.928,A -85,B 0,C 180,E1 -17390.681,E2 -17390.681} C_VEL
LIN {X 0,Y 284.603,Z 495.688,A -85,B 0,C 180,E1 -17391.55,E2 -17391.55} C_VEL
LIN {X 0,Y 284.05,Z 487.11,A -85,B 0,C 180,E1 -17392.719,E2 -17392.719} C_VEL
LIN {X 0,Y 282.998,Z 477.379,A -85,B 0,C 180,E1 -17393.869,E2 -17393.869} C_VEL
LIN {X 0,Y 281.302,Z 467.7,A -85,B 0,C 180,E1 -17394.876,E2 -17394.876} C_VEL
LIN {X 0,Y 278.75,Z 457.037,A -85,B 0,C 180,E1 -17395.845,E2 -17395.845} C_VEL
LIN {X 0,Y 276.221,Z 447.896,A -85,B 0,C 180,E1 -17396.554,E2 -17396.554} C_VEL
LIN {X 0,Y 276.179,Z 447.325,A -85,B 0,C 180,E1 -17396.583,E2 -17396.583} C_VEL
LIN {X 0,Y 276.672,Z 443.567,A -85,B 0,C 180,E1 -17400.532,E2 -17400.532} C_VEL
LIN {X 0,Y 277.153,Z 440.534,A -85,B 0,C 180,E1 -17403.908,E2 -17403.908} C_VEL
LIN {X 0,Y 277.715,Z 437.502,A -85,B 0,C 180,E1 -17407.398,E2 -17407.398} C_VEL
LIN {X 0,Y 278.182,Z 434.496,A -85,B 0,C 180,E1 -17411.06,E2 -17411.06} C_VEL
LIN {X 0,Y 278.311,Z 432.991,A -85,B 0,C 180,E1 -17412.984,E2 -17412.984} C_VEL
LIN {X 0,Y 278.322,Z 431.493,A -85,B 0,C 180,E1 -17415.005,E2 -17415.005} C_VEL
LIN {X 0,Y 278.017,Z 428.799,A -85,B 0,C 180,E1 -17418.908,E2 -17418.908} C_VEL
LIN {X 0,Y 277.653,Z 426.493,A -85,B 0,C 180,E1 -17422.591,E2 -17422.591} C_VEL
LIN {X 0,Y 277.346,Z 424.149,A -85,B 0,C 180,E1 -17426.742,E2 -17426.742} C_VEL
LIN {X 0,Y 277.249,Z 423.58,A -85,B 0,C 180,E1 -17427.836,E2 -17427.836} C_VEL
LIN {X 0,Y 277.287,Z 423.446,A -85,B 0,C 180,E1 -17431.211,E2 -17431.211} C_VEL
LIN {X 0,Y 277.306,Z 423.443,A -85,B 0,C 180,E1 -17434.478,E2 -17434.478} C_VEL
LIN {X 0,Y 277.264,Z 423.45,A -85,B 0,C 180,E1 -17437.652,E2 -17437.652} C_VEL
LIN {X 0,Y 277.338,Z 423.437,A -85,B 0,C 180,E1 -17440.765,E2 -17440.765} C_VEL
LIN {X 0,Y 277.423,Z 423.428,A -85,B 0,C 180,E1 -17445.324,E2 -17445.324} C_VEL
LIN {X 0,Y 277.456,Z 423.425,A -85,B 0,C 180,E1 -17449.786,E2 -17449.786} C_VEL
LIN {X 0,Y 277.635,Z 423.399,A -85,B 0,C 180,E1 -17452.728,E2 -17452.728} C_VEL
LIN {X 0,Y 277.815,Z 423.375,A -85,B 0,C 180,E1 -17458.55,E2 -17458.55} C_VEL
LIN {X 0,Y 277.815,Z 423.365,A -85,B 0,C 180,E1 -17461.449,E2 -17461.449} C_VEL
LIN {X 0,Y 277.634,Z 423.404,A -85,B 0,C 180,E1 -17467.271,E2 -17467.271} C_VEL
LIN {X 0,Y 277.455,Z 423.42,A -85,B 0,C 180,E1 -17470.212,E2 -17470.212} C_VEL
LIN {X 0,Y 277.421,Z 423.424,A -85,B 0,C 180,E1 -17474.674,E2 -17474.674} C_VEL
LIN {X 0,Y 277.338,Z 423.436,A -85,B 0,C 180,E1 -17479.233,E2 -17479.233} C_VEL
LIN {X 0,Y 277.312,Z 423.438,A -85,B 0,C 180,E1 -17484.17,E2 -17484.17} C_VEL
LIN {X 0,Y 277.319,Z 423.44,A -85,B 0,C 180,E1 -17487.505,E2 -17487.505} C_VEL
LIN {X 0,Y 277.266,Z 423.447,A -85,B 0,C 180,E1 -17490.481,E2 -17490.481} C_VEL
LIN {X 0,Y 277.248,Z 423.448,A -85,B 0,C 180,E1 -17493.895,E2 -17493.895} C_VEL
LIN {X 0,Y 277.28,Z 423.444,A -85,B 0,C 180,E1 -17497.466,E2 -17497.466} C_VEL
LIN {X 0,Y 277.286,Z 423.445,A -85,B 0,C 180,E1 -17501.221,E2 -17501.221} C_VEL
LIN {X 0,Y 277.237,Z 423.451,A -85,B 0,C 180,E1 -17505.218,E2 -17505.218} C_VEL
LIN {X 0,Y 277.22,Z 423.451,A -85,B 0,C 180,E1 -17509.511,E2 -17509.511} C_VEL
LIN {X 0,Y 277.276,Z 423.448,A -85,B 0,C 180,E1 -17512.533,E2 -17512.533} C_VEL
LIN {X 0,Y 277.249,Z 423.45,A -85,B 0,C 180,E1 -17516.105,E2 -17516.105} C_VEL
LIN {X 0,Y 277.256,Z 423.448,A -85,B 0,C 180,E1 -17519.539,E2 -17519.539} C_VEL
LIN {X 0,Y 277.35,Z 423.437,A -85,B 0,C 180,E1 -17523.179,E2 -17523.179} C_VEL
LIN {X 0,Y 278.418,Z 426.397,A -85,B 0,C 180,E1 -17523.394,E2 -17523.394} C_VEL
LIN {X 0,Y 284.607,Z 439.727,A -85,B 0,C 180,E1 -17524.535,E2 -17524.535} C_VEL
LIN {X 0,Y 289.327,Z 448.309,A -85,B 0,C 180,E1 -17525.489,E2 -17525.489} C_VEL
LIN {X 0,Y 295.668,Z 457.765,A -85,B 0,C 180,E1 -17526.765,E2 -17526.765} C_VEL
LIN {X 0,Y 303.985,Z 468.255,A -85,B 0,C 180,E1 -17528.429,E2 -17528.429} C_VEL
LIN {X 0,Y 313.39,Z 478.914,A -85,B 0,C 180,E1 -17530.367,E2 -17530.367} C_VEL
LIN {X 0,Y 319.828,Z 485.852,A -85,B 0,C 180,E1 -17531.874,E2 -17531.874} C_VEL
LIN {X 0,Y 325.482,Z 491.689,A -85,B 0,C 180,E1 -17533.305,E2 -17533.305} C_VEL
LIN {X 0,Y 331.337,Z 497.264,A -85,B 0,C 180,E1 -17534.94,E2 -17534.94} C_VEL
LIN {X 0,Y 335.951,Z 501.44,A -85,B 0,C 180,E1 -17536.377,E2 -17536.377} C_VEL
LIN {X 0,Y 340.773,Z 505.986,A -85,B 0,C 180,E1 -17538.098,E2 -17538.098} C_VEL
LIN {X 0,Y 344.215,Z 508.707,A -85,B 0,C 180,E1 -17539.412,E2 -17539.412} C_VEL
LIN {X 0,Y 347.066,Z 510.958,A -85,B 0,C 180,E1 -17540.677,E2 -17540.677} C_VEL
LIN {X 0,Y 349.147,Z 513.102,A -85,B 0,C 180,E1 -17541.9,E2 -17541.9} C_VEL
LIN {X 0,Y 351.041,Z 514.833,A -85,B 0,C 180,E1 -17543.101,E2 -17543.101} C_VEL
LIN {X 0,Y 353.043,Z 516.234,A -85,B 0,C 180,E1 -17544.461,E2 -17544.461} C_VEL
LIN {X 0,Y 354.345,Z 516.997,A -85,B 0,C 180,E1 -17545.45,E2 -17545.45} C_VEL
LIN {X 0,Y 355.709,Z 517.556,A -85,B 0,C 180,E1 -17546.602,E2 -17546.602} C_VEL
LIN {X 0,Y 356.759,Z 517.857,A -85,B 0,C 180,E1 -17547.742,E2 -17547.742} C_VEL
LIN {X 0,Y 357.455,Z 517.969,A -85,B 0,C 180,E1 -17548.873,E2 -17548.873} C_VEL
LIN {X 0,Y 357.661,Z 518.027,A -85,B 0,C 180,E1 -17550,E2 -17550} C_VEL
LIN {X 0,Y 357.419,Z 517.996,A -85,B 0,C 180,E1 -17551.127,E2 -17551.127} C_VEL
LIN {X 0,Y 356.749,Z 517.859,A -85,B 0,C 180,E1 -17552.258,E2 -17552.258} C_VEL
LIN {X 0,Y 355.709,Z 517.551,A -85,B 0,C 180,E1 -17553.398,E2 -17553.398} C_VEL
LIN {X 0,Y 354.364,Z 516.992,A -85,B 0,C 180,E1 -17554.55,E2 -17554.55} C_VEL
